(* Logix 5000 project; controller CLASE_1 Emulate 5570 rev 28.11; software revision 28.02; part 8 of 15 *)
(* tags used below, declared in another part *)
   Inp_PosFdbk : REAL;   // Position Feedback from Valve (in Raw Input units)
   Inp_OpenLS : BOOL;   // Valve Open Limit Switch 1=confirmed fully open
   Inp_ClosedLS : BOOL;   // Valve Closed Limit Switch 1=confirmed fully closed
   Inp_ActuatorFault : BOOL;   // Valve Actuator Fault (overload, etc.), 0=OK, 1=Fault)
   Inp_IntlkOK : BOOL;   // 1=Interlocks OK, Pulse Output Valve can be moved
   Inp_NBIntlkOK : BOOL;   // 1=Non-Bypassable Interlocks OK, Pulse Output Valve can be moved
   Inp_IOFault : BOOL;   // Input / Output Communication Status 0=OK, 1=fail
   Inp_Sim : BOOL;   // 1=I/O are being simulated, set output CV to 0.0, ignore I/O Fault
   Inp_OvrdCV : REAL;   // CV target in Override Mode (CV EU)
   Inp_Reset : BOOL;   // 1=Reset latched Alarms
   Cfg_ShedHold : BOOL;   // 1=Hold Output on Interlock or bad PV, 0=Go to Cfg_IntlkCV
   Cfg_ShedOnIOFault : BOOL;   // 1=Take shed action (hold or interlock CV) on I/O Fault
   Cfg_SkipRoCLim : BOOL;   // 1=Skip RoC Limiting in Intlk, Maint, Ovrd modes
   Cfg_SetTrack : BOOL;   // 1=PSets track OSets in Oper, OSets track PSets in Prog, 0=no tracking
   Cfg_SetTrackOvrdHand : BOOL;   // 1=Prog/Oper Settings track Override/Hand CV
   Cfg_HasOpenLS : BOOL;   // 1=Valve provides an Open Limit Switch signal
   Cfg_HasClosedLS : BOOL;   // 1=Valve provides a Closed Limit Switch signal
   Cfg_UseOpenLS : BOOL;   // 1=Valve Open LS should be used for open/closed status
   Cfg_UseClosedLS : BOOL;   // 1=Valve Closed LS should be used for open/closed status
   Cfg_LSFail : BOOL;   // 1=both switches ON=fail, 0=both switches OFF=fail
   Cfg_PCmdClear : ALIAS FOR Mode.Cfg_PCmdClear;
   Cfg_OvrdIntlk : BOOL;   // 1=Override ignores Bypassable Intlk; 0=always use Intlk
   Cfg_MinCV : REAL;   // Minimum CV (in CV EU, for limiting)
   Cfg_MaxCV : REAL;   // Maximum CV (in CV EU, for limiting)
   Cfg_MaxCVRoCInc : REAL;   // Maximum allowed CV Rate of Change (Increasing) Setting (EU/sec)
   Cfg_MaxCVRoCDec : REAL;   // Maximum allowed CV Rate of Change (Decreasing) Setting (EU/sec)
   Cfg_IntlkCV : REAL;   // CV (target in EU) when interlocked (if not Cfg_ShedHold)
   Cfg_CVEUMin : REAL;   // CV Minimum in Engineering Units (for scaling)
   Cfg_CVEUMax : REAL;   // CV Maximum in Engineering Units (for scaling)
   Cfg_CVRawMin : REAL;   // CV Minimum in I/O (raw) Units (for scaling)
   Cfg_CVRawMax : REAL;   // CV Maximum in I/O (raw) Units (for scaling)
   Cfg_FdbkRawMin : REAL;   // Position Feedback Minimum in raw input units (for scaling)
   Cfg_FdbkRawMax : REAL;   // Position Feedback Maximum in raw input units (for scaling)
   Cfg_CycleT : REAL;   // Open and Close Pulse Output overall period (s)
   Cfg_OpenRate : REAL;   // Rate at which valve moves when opening (CV EU/sec)
   Cfg_CloseRate : REAL;   // Rate at which valve moves when closing (CV EU/sec)
   Cfg_MaxOnT : REAL;   // Open and Close Pulse Output maximum ON time (s)
   Cfg_MinOnT : REAL;   // Open and Close Pulse Output minimum ON time (s)
   Cfg_BumpT : REAL;   // Time to bump valve open or closed (by Oper) when Fdbk Bad (sec)
   Cfg_Deadtime : REAL;   // Additional time on first pulse after stop or direction change
   Cfg_MaxClosedPos : REAL;   // Position above which valve is assumed open if limit switches not used
   PSet_CV : REAL;   // Program Setting of Controlled Variable (output) (CV EU)
   PSet_CVRoCLimInc : REAL;   // Program Setting of CV Rate of Change Limit, Increasing, (in EU/sec)
   PSet_CVRoCLimDec : REAL;   // Program Setting of CV Rate of Change Limit, Decreasing, (in EU/sec)
   PSet_Owner : DINT;   // Program Owner Request ID (non-zero) or Release (zero)
   OSet_CV : REAL;   // Operator Setting of Controlled Variable (output) (CV EU)
   OSet_CVRoCLimInc : REAL;   // Operator Setting of CV Rate of Change Limit, Increasing, (in EU/sec)
   OSet_CVRoCLimDec : REAL;   // Operator Setting of CV Rate of Change Limit, Decreasing, (in EU/sec)
   PCmd_Reset : BOOL;   // Program Command to Reset Alarms requiring Reset
   OCmd_BumpOpen : BOOL;   // Operator Command to bump valve open (avail. if Fdbk Bad)
   OCmd_BumpClose : BOOL;   // Operator Command to bump valve closed (avail. if Fdbk Bad)
   OCmd_Bypass : BOOL;   // Operator Command to Bypass all Bypassable Interlocks
   OCmd_Check : BOOL;   // Operator Command to Check (not bypass) all Interlocks
   MCmd_Disable : BOOL;   // Maintenance Command to Pulse Output Valve
   MCmd_Enable : BOOL;   // Maintenance Command to Enable Pulse Output Valve
   OCmd_Reset : BOOL;   // Operator Command to Reset all Alarms requiring Reset
   OCmd_ResetAckAll : BOOL;   // Operator Command to Reset all Alarms and latched Shed conditions
   Out_CV : REAL;   // CV Output in Raw (I/O Card) Units
   Val_Pos : REAL;   // Valve actual position from feedback (CV EU)
   Val_CVOut : REAL;   // Value of CV output (after clamping and ramping) (CV EU)
   Val_CVEUMin : REAL;   // Minimum of scaled range = MIN (Cfg_CVEUMin, Cfg_CVEUMax)
   Val_CVEUMax : REAL;   // Maximum of scaled range = MAX (Cfg_CVEUMin, Cfg_CVEUMax)
   SrcQ_IO : SINT;   // Source and Quality of primary I/O (enumeration)
   SrcQ : SINT;   // Source and Quality of primary Val/Sts (enumeration)
   Val_Fdbk : SINT;   // Device Feedback 0=Moving, 1=Closed, 2=Opened, 3=Limit Switch Failure
   Val_Sts : SINT;   // 0=AtTarget, 1=RampClose, 2=RampOpen, 3=Clamp@Min, 4=Clamp@Max, 5=BumpClose, 6=BumpOpen, 33=Disabled
   Val_Owner : DINT;   // Current Object Owner ID (0=not owned)
   Sts_CVInfNaN : BOOL;   // 1=Selected CV is Infinite or Not A Number (1.$, 1.#NaN)
   Sts_PosInfNaN : BOOL;   // 1=Inp_PosFdbk is Infinite or Not A Number (1.$, 1.#NaN)
   Sts_Ramping : BOOL;   // 1=CV is ramping to target
   Sts_Clamped : BOOL;   // 1=CV Set is clamped at CVMin or CVMax
   Sts_SkipRoCLim : BOOL;   // 1=Rate of Change Limiting was skipped this scan (Maint, Ovrd, Intlk, Hand)
   Sts_Active : BOOL;   // 1=CV is greater than Cfg_MaxClosedPos, show valve symbol as "opened"
   Sts_Available : BOOL;   // 1=Pulse Output Valve available for control by automation (Prog)
   Sts_Bypass : BOOL;   // 1=Bypassable Interlocks are Bypassed
   Sts_BypActive : BOOL;   // 1=Bypassing Active (Bypassed or Maintenance)
   Sts_Disabled : BOOL;   // 1=Output is Disabled
   Sts_LSFail : BOOL;   // 1=Limit Switch Overlap Failure
   Sts_NotRdy : BOOL;   // 1=Device Not Ready, see detail bits for reason
   Nrdy_Disabled : BOOL;   // 1=Device Not Ready: Device Disabled by Maintenance
   Nrdy_CfgErr : BOOL;   // 1=Device Not Ready: Configuration Error
   Nrdy_Intlk : BOOL;   // 1=Device Not Ready: Interlock Not OK
   Nrdy_IOFault : BOOL;   // 1=Device Not Ready: I/O Fault (Shed Requires Reset)
   Nrdy_NoMode : BOOL;   // 1=Device Not Ready: Device Logic Disabled / NO Mode
   Sts_MaintByp : BOOL;   // 1=Device has a Maintenance Bypass function active
   Sts_Err : BOOL;   // 1=Error in Config: see detail bits for reason
   Err_Limit : BOOL;   // 1=Error in Config: CV Limits swapped
   Err_EU : BOOL;   // 1=Error in Config: Scaled CV EU Min = Max
   Err_Raw : BOOL;   // 1=Error in Config: Raw Output Scaling Min = Max
   Err_Fdbk : BOOL;   // 1=Error in Config: Raw Feedback Scaling Min = Max
   Err_Timer : BOOL;   // 1=Error in Config: Invalid Timer Preset (use 0 to 2147483)
   Err_Alarm : BOOL;   // 1=Error in Config: Alarm Min On Time, Shelf Time, Severity
   Sts_Hand : ALIAS FOR Mode.Sts_Hand;
   Sts_Maint : ALIAS FOR Mode.Sts_Maint;
   Sts_Ovrd : ALIAS FOR Mode.Sts_Ovrd;
   Sts_Prog : ALIAS FOR Mode.Sts_Prog;
   Sts_Oper : ALIAS FOR Mode.Sts_Oper;
   Sts_IntlkTrip : ALIAS FOR IntlkTrip.Inp;   // 1=Status: CV held or forced by interlock NOT OK (1-shot)
   Sts_ActuatorFault : ALIAS FOR ActuatorFault.Inp;   // 1=Actuator Fault detected (input)
   Sts_IOFault : ALIAS FOR IOFault.Inp;   // 1=I/O Fault Status (0=OK, 1=Bad)
   Rdy_BumpOpen : BOOL;   // 1=Ready to receive OCmd_BumpOpen (enables HMI button)
   Rdy_BumpClose : BOOL;   // 1=Ready to receive OCmd_BumpClose (enables HMI button)
   Rdy_Bypass : BOOL;   // 1=Ready to receive OCmd_Bypass (enables HMI button)
   Rdy_Check : BOOL;   // 1=Ready to receive OCmd_Check (enables HMI button)
   Rdy_Disable : BOOL;   // 1=Ready to receive MCmd_Disable (enables HMI button)
   Rdy_Enable : BOOL;   // 1=Ready to receive MCmd_Enable (enables HMI button)
   Rdy_CV : BOOL;   // 1=Ready to receive OSet_CV (enables data entry field)
   Rdy_CVRoCLimInc : BOOL;   // 1=Ready to receive OSet_CVRoCLimInc (enables data entry field)
   Rdy_CVRoCLimDec : BOOL;   // 1=Ready to receive OSet_CVRoCLimDec (enables data entry field)
   P_ValveC : BOOL;   // Unique Parameter Name for auto - discovery
   Mode : P_Mode;   // Pulse Output Valve Mode Selection
   IOFault : P_Alarm;   // I/O Fault Alarm
   IntlkTrip : P_Alarm;   // Interlock Trip Alarm
   Cfg_Tag : STRING_20;   // Tagname for display on HMI
   Cfg_Label : STRING_20;   // Label for graphic symbol displayed on HMI
   Cfg_Desc : STRING_40;   // Description for display on HMI
   Wrk_Bypass : BOOL;   // Internal Bypassable Interlocks are Bypassed flag
   Wrk_Disabled : BOOL;   // Internal Pulse Output Valve Disabled status
   Cfg_EU : STRING_8;   // Engineering Units for display on HMI
   Wrk_CV : REAL;   // Working copy of Speed Reference (for limiting)
   Wrk_CVRoCLimInc : REAL;   // Selected CV Rate of Change Limit Increasing
   Wrk_CVSet : REAL;   // Final selected CV to feed to RoC Limiter
   Wrk_CVOut : REAL;   // Working value of CV after Rate Limiting
   Wrk_IntlkTripONS : BOOL;   // Interlock Tripped This Scan
   Wrk_ScanTime : REAL;   // Seconds since previous scan
   Wrk_StepInc : REAL;   // Amount to increase CV (to valve pulse logic) this scan for rate limiting
   Wrk_ScanT : TIMER;   // Scan Timer (milliseconds, always runs)
   ActuatorFault : P_Alarm;   // Actuator Fault Alarm (based on Actuator Fault Input)
   Wrk_RealChkDINT : DINT;   // REAL tag bit pattern as a DINT to check for Inf / NaN
   Wrk_Close : BOOL;   // Internal Close output -- before Sim
   Wrk_Open : BOOL;   // Internal Open output -- before Sim
   Wrk_CycleT : TIMER;   // Overall Cycle Timer for pulsed outputs
   Wrk_OKtoOpen : BOOL;   // OK to pulse Out_Open
   Wrk_OKtoClose : BOOL;   // OK to pulse Out_Close
   Wrk_OpenTime : REAL;   // Time to pulse Out_Open
   Wrk_CycleT_ms : DINT;   // Cycle Time in milliseconds (preset)
   Wrk_CloseTime : REAL;   // Time to pulse Out_Close
   Inf_Type : STRING_16;   // Must contain AOI name, used for HMI and Information S/W
   Wrk_OpenFdbk : BOOL;   // 1=LS Feedback shows valve confirmed open
   Wrk_ClosedFdbk : BOOL;   // 1=LS Feedback shows valve confirmed closed
   Wrk_StepDec : REAL;   // Amount to decrease CV (to valve pulse logic) this scan for rate limiting
   Wrk_CVRoCLimDec : REAL;   // Selected CV Rate of Change Limit Decreasing
   Wrk_BumpClose : BOOL;   // Operator Bump Close requested
   Wrk_BumpOpen : BOOL;   // Operator Bump Open requested
   Wrk_BumpingOpen : BOOL;   // Operator Bump Open actively pulsing Out_Open
   Wrk_BumpingClose : BOOL;   // Operator Bump Close actively pulsing Out_Close
   Inf_Lib : STRING_12;   // Display Library for Faceplate call-up
   Cfg_CVNavTag : STRING_NavTag;   // Tagname for destination of CV Navigation button
   Wrk_ShedIntlkCV : BOOL;   // Output CV being held at Interlock value
   Wrk_ShedHold : BOOL;   // Output CV being held at last good value
(* P_ValveC, continued *)

ROUTINE Logic   (* ladder *)
// Normal Scan: control Analog Output
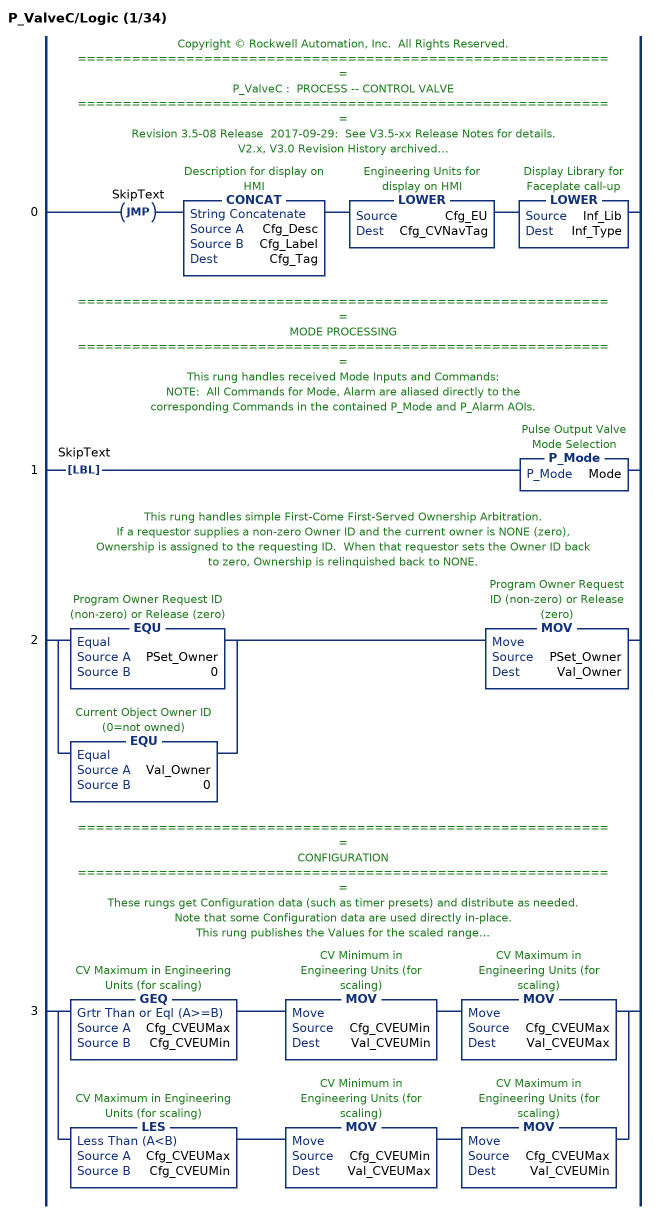
   // Copyright © Rockwell Automation, Inc.  All Rights Reserved.
   // ============================================================
   // P_ValveC :  PROCESS -- CONTROL VALVE
   // ============================================================
   // Revision 3.5-08 Release  2017-09-29:  See V3.5-xx Release Notes for details.
   // V2.x, V3.0 Revision History archived.
   // V3.1-00  2014-07-22:  Modified to use P_Alarm, P_Mode V3.1; added
   // Not Ready reason bits (Nrdy_Xxxxx), source/quality values (SrcQ).
   // Modified to consistently use alias tag names.  Added check for
   // Err_Fdbk on scaling of position feedback.
   // V3.1-01  2014-09-03:  Corrections to Nrdy_ resets. Modified logic for
   // Err_Fdbk. Using P_Alarm, P_Mode V3.1-01.
   // V3.1-02  2014-09-30:  Unchanged, but using P_Alarm V3.1-02.
   // V3.1-03  2015-01-21:  Corrected Maintenance Bypass indication for limit switches.
   // Modified to prevent output pulsing on additional fault conditions.
   //  Modified to show Val_Sts = 1 or 2 when moving via pulsing.
   // V3.1-04 Patch01  2015-09-25: Modified Err_Fdbk, Err_Raw, handling of Cfg_CycleT.
   // V3.5-01  2016-01-29:  Unchanged, but using P_Alarm V3.5-01.
   // V3.5-03 Patch01  2016-07-06:  Modified logic which triggers IntlkTrip status/alarm.
   // V3.5-05  2016-12-16:   Changed Nav Tags to user-defined STRING_NavTag type.
   // V3.5-08  2017-09-29:  Modified CV Rate of Change handling for limits = 0.0 (unlimited).
   // ============================================================
   // This Instruction controls a Pulse Output Valve with
   // analog position feedback and provides:
   // *  Program and Operator entry of target position in Percent Open
   // *  Ramping of position to target at specified Rate of Change (%/sec)
   // *  Scaling of Position Feedback input from Raw (I/O card) Units to percent
   // *  Monitoring of Interlock conditions which cause output to shed
   // *  Configurable shed to HOLD or to configured position
   // *  Monitoring of I/O communication faults
   // *  Alarms for Interlock Trip, Actuator Fault, I/O Fault
   // *  Opened, Closed status based on limit switches (if provided),
   // or based on Position Feedback and a configured threshold.
   // *  "Available" status for use by automation logic to know whether valve
   //       can be controlled by other objects.
   // Modes are provided by a P_Mode AOI instance.
   // Alarms are provided by P_Alarm AOI instances.
   // Modes of operation: Operator, Program, Override, Maintenance, Hand
   // ============================================================
   // SHOW LOCAL STRINGS
   // ============================================================
   // The STRINGs containing the text associated with each instance of this
   // instruction cannot be Input or Output Parameters, because STRINGs are not
   //  'atomic' types. (Inputs and Outputs must be SINT, INT, DINT, REAL, or BOOL.)
   // In order to make it easier to find and configure these STRINGs, this rung
   // was added.  THE JMP (and the LBL on the following rung)
   // MUST NOT BE REMOVED!!!
   // To view the STRINGs, go to the instruction instance (in LD or FBD), RIGHT-click
   // to bring up the context menu and select "Open Instruction Logic".
   // This rung will appear with the STRING values for the selected instance.
   // You may double-click the STRING values here to modify them as well.
   // #####  V3.1-00  2014-07-15: Added Cfg_CVNavTag to displayed strings  #####
   0: JMP(SkipText)CONCAT(Cfg_Desc,Cfg_Label,Cfg_Tag)LOWER(Cfg_EU,Cfg_CVNavTag)LOWER(Inf_Lib,Inf_Type);
   // ============================================================
   // MODE PROCESSING
   // ============================================================
   // This rung handles received Mode Inputs and Commands:
   // NOTE:  All Commands for Mode, Alarm are aliased directly to the
   // corresponding Commands in the contained P_Mode and P_Alarm AOIs.
   1: LBL(SkipText)P_Mode(Mode);
   // This rung handles simple First-Come First-Served Ownership Arbitration.
   // If a requestor supplies a non-zero Owner ID and the current owner is NONE (zero),
   // Ownership is assigned to the requesting ID.  When that requestor sets the Owner ID back
   // to zero, Ownership is relinquished back to NONE.
   2: [EQU(PSet_Owner,0) ,EQU(Val_Owner,0) ]MOV(PSet_Owner,Val_Owner);
   // ============================================================
   // CONFIGURATION
   // ============================================================
   // These rungs get Configuration data (such as timer presets) and distribute as needed.
   // Note that some Configuration data are used directly in-place.
   // This rung publishes the Values for the scaled range.
   // If this instruction is reverse scaled by reversing the scaled (EU) min and max configurations,
   // the values are swapped so the the EUMax Value is always greater than the EUMin Value.
   // This makes the HMI bargraph and trend coding easier, and provides values
   // that can be pinned to the CV EU configuration of a PID, so the AOut and PID ranges are in lockstep.
   3: [GEQ(Cfg_CVEUMax,Cfg_CVEUMin) MOV(Cfg_CVEUMin,Val_CVEUMin) MOV(Cfg_CVEUMax,Val_CVEUMax) ,LES(Cfg_CVEUMax,Cfg_CVEUMin) MOV(Cfg_CVEUMin,Val_CVEUMax) MOV(Cfg_CVEUMax,Val_CVEUMin) ];
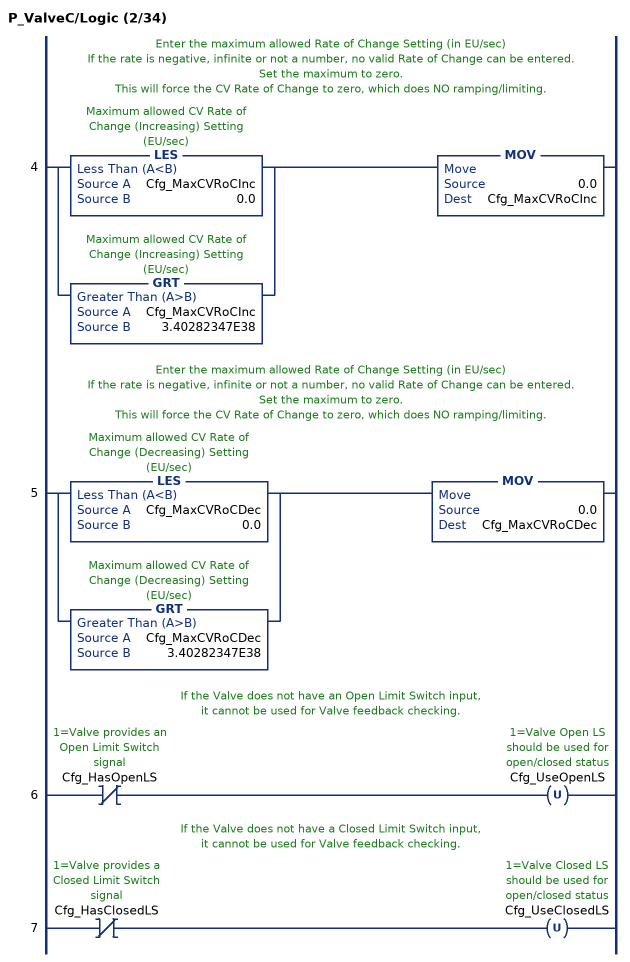
   // Enter the maximum allowed Rate of Change Setting (in EU/sec)
   // If the rate is negative, infinite or not a number, no valid Rate of Change can be entered.  Set the maximum to zero.
   // This will force the CV Rate of Change to zero, which does NO ramping/limiting.
   4: [LES(Cfg_MaxCVRoCInc,0.0) ,GRT(Cfg_MaxCVRoCInc,3.40282347E38) ]MOV(0.0,Cfg_MaxCVRoCInc);
   // Enter the maximum allowed Rate of Change Setting (in EU/sec)
   // If the rate is negative, infinite or not a number, no valid Rate of Change can be entered.  Set the maximum to zero.
   // This will force the CV Rate of Change to zero, which does NO ramping/limiting.
   5: [LES(Cfg_MaxCVRoCDec,0.0) ,GRT(Cfg_MaxCVRoCDec,3.40282347E38) ]MOV(0.0,Cfg_MaxCVRoCDec);
   // If the Valve does not have an Open Limit Switch input,
   // it cannot be used for Valve feedback checking.
   6: XIO(Cfg_HasOpenLS)OTU(Cfg_UseOpenLS);
   // If the Valve does not have a Closed Limit Switch input,
   // it cannot be used for Valve feedback checking.
   7: XIO(Cfg_HasClosedLS)OTU(Cfg_UseClosedLS);
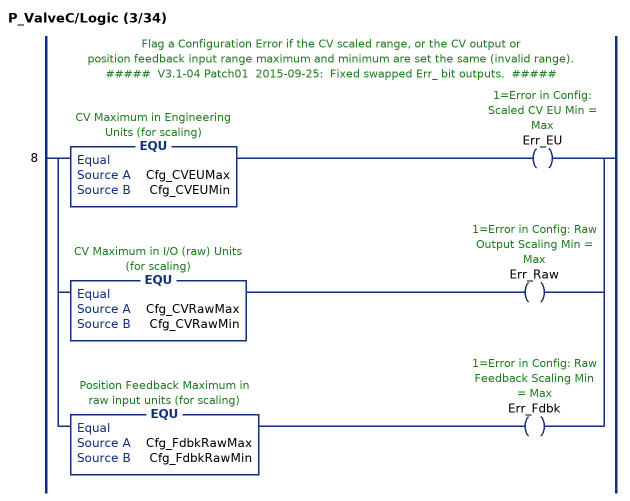
   // Flag a Configuration Error if the CV scaled range, or the CV output or
   // position feedback input range maximum and minimum are set the same (invalid range).
   // #####  V3.1-04 Patch01  2015-09-25:  Fixed swapped Err_ bit outputs.  #####
   8: [EQU(Cfg_CVEUMax,Cfg_CVEUMin) OTE(Err_EU) ,EQU(Cfg_CVRawMax,Cfg_CVRawMin) OTE(Err_Raw) ,EQU(Cfg_FdbkRawMax,Cfg_FdbkRawMin) OTE(Err_Fdbk) ];
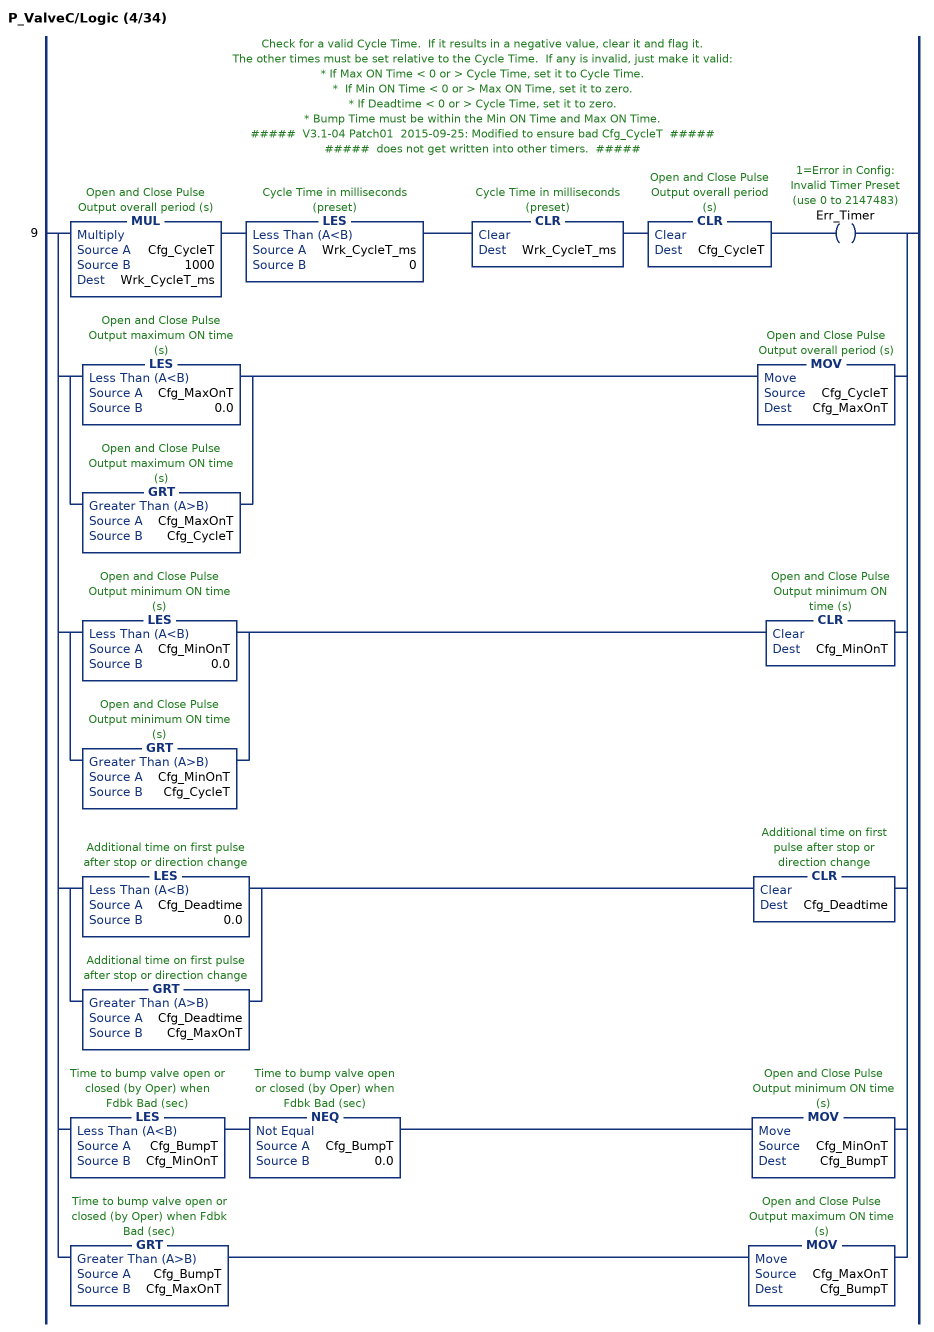
   // Check for a valid Cycle Time.  If it results in a negative value, clear it and flag it.
   // The other times must be set relative to the Cycle Time.  If any is invalid, just make it valid:
   // * If Max ON Time < 0 or > Cycle Time, set it to Cycle Time.
   // *  If Min ON Time < 0 or > Max ON Time, set it to zero.
   // * If Deadtime < 0 or > Cycle Time, set it to zero.
   // * Bump Time must be within the Min ON Time and Max ON Time.
   // #####  V3.1-04 Patch01  2015-09-25: Modified to ensure bad Cfg_CycleT  #####
   // #####  does not get written into other timers.  #####
   9: [MUL(Cfg_CycleT,1000,Wrk_CycleT_ms) LES(Wrk_CycleT_ms,0) CLR(Wrk_CycleT_ms) CLR(Cfg_CycleT) OTE(Err_Timer) ,[LES(Cfg_MaxOnT,0.0) ,GRT(Cfg_MaxOnT,Cfg_CycleT) ] MOV(Cfg_CycleT,Cfg_MaxOnT) ,[LES(Cfg_MinOnT,0.0) ,GRT(Cfg_MinOnT,Cfg_CycleT) ] CLR(Cfg_MinOnT) ,[LES(Cfg_Deadtime,0.0) ,GRT(Cfg_Deadtime,Cfg_MaxOnT) ] CLR(Cfg_Deadtime) ,LES(Cfg_BumpT,Cfg_MinOnT) NEQ(Cfg_BumpT,0.0) MOV(Cfg_MinOnT,Cfg_BumpT) ,GRT(Cfg_BumpT,Cfg_MaxOnT) MOV(Cfg_MaxOnT,Cfg_BumpT) ];
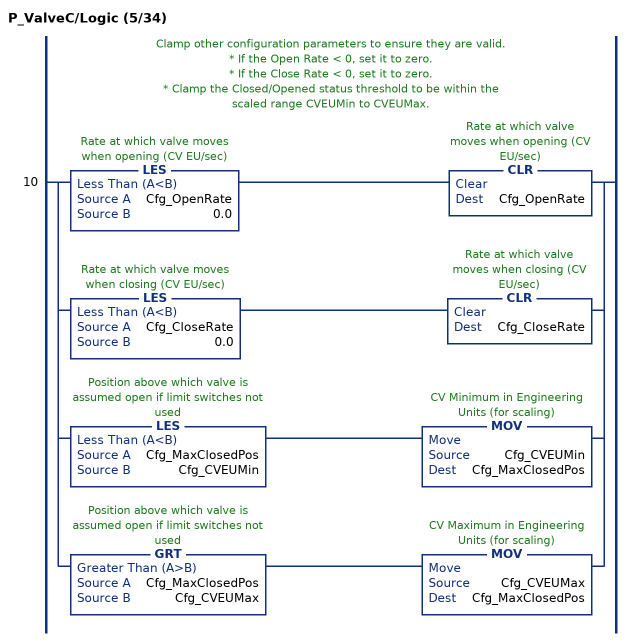
   // Clamp other configuration parameters to ensure they are valid.
   // * If the Open Rate < 0, set it to zero.
   // * If the Close Rate < 0, set it to zero.
   // * Clamp the Closed/Opened status threshold to be within the
   // scaled range CVEUMin to CVEUMax.
   10: [LES(Cfg_OpenRate,0.0) CLR(Cfg_OpenRate) ,LES(Cfg_CloseRate,0.0) CLR(Cfg_CloseRate) ,LES(Cfg_MaxClosedPos,Cfg_CVEUMin) MOV(Cfg_CVEUMin,Cfg_MaxClosedPos) ,GRT(Cfg_MaxClosedPos,Cfg_CVEUMax) MOV(Cfg_CVEUMax,Cfg_MaxClosedPos) ];
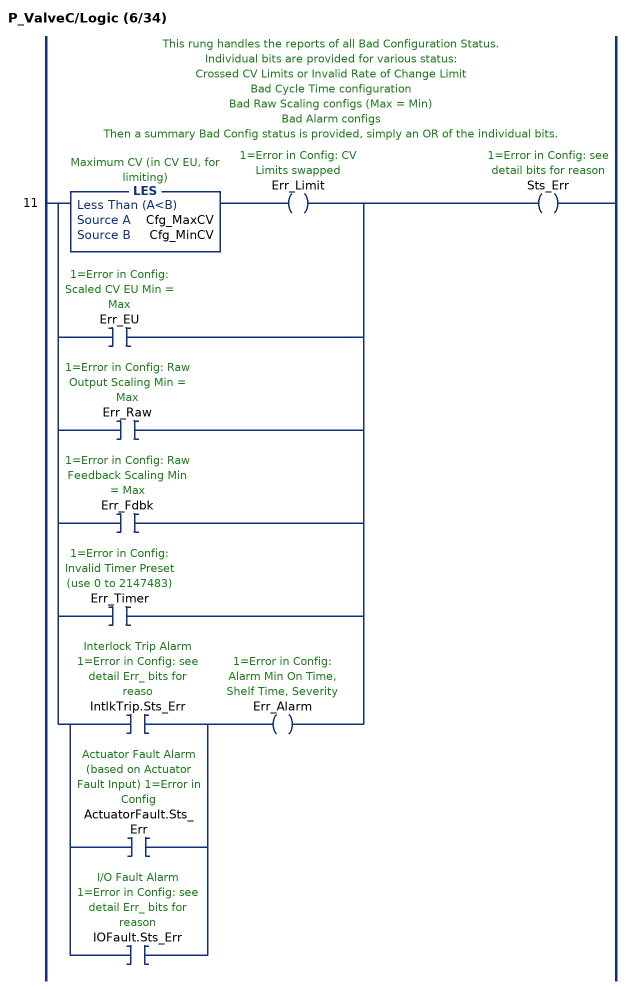
   // This rung handles the reports of all Bad Configuration Status.
   // Individual bits are provided for various status:
   // Crossed CV Limits or Invalid Rate of Change Limit
   // Bad Cycle Time configuration
   // Bad Raw Scaling configs (Max = Min)
   // Bad Alarm configs
   // Then a summary Bad Config status is provided, simply an OR of the individual bits.
   11: [LES(Cfg_MaxCV,Cfg_MinCV) OTE(Err_Limit) ,XIC(Err_EU) ,XIC(Err_Raw) ,XIC(Err_Fdbk) ,XIC(Err_Timer) ,[XIC(IntlkTrip.Sts_Err) ,XIC(ActuatorFault.Sts_Err) ,XIC(IOFault.Sts_Err) ] OTE(Err_Alarm) ]OTE(Sts_Err);
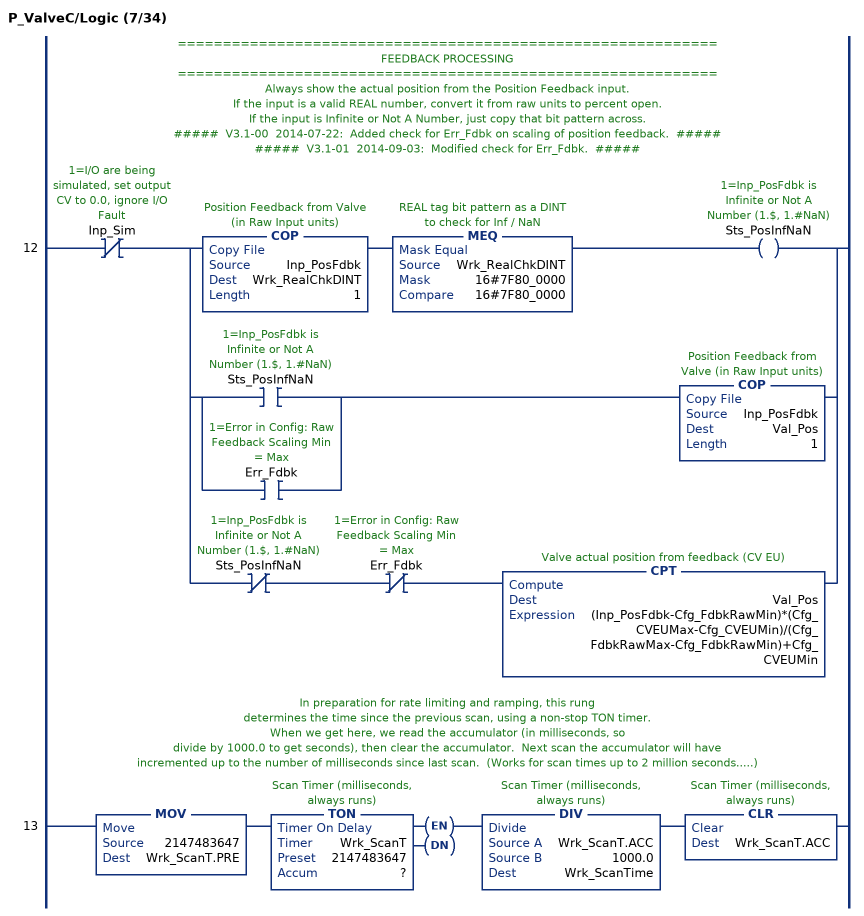
   // ============================================================
   // FEEDBACK PROCESSING
   // ============================================================
   // Always show the actual position from the Position Feedback input.
   // If the input is a valid REAL number, convert it from raw units to percent open.
   // If the input is Infinite or Not A Number, just copy that bit pattern across.
   // #####  V3.1-00  2014-07-22:  Added check for Err_Fdbk on scaling of position feedback.  #####
   // #####  V3.1-01  2014-09-03:  Modified check for Err_Fdbk.  #####
   12: XIO(Inp_Sim)[COP(Inp_PosFdbk,Wrk_RealChkDINT,1) MEQ(Wrk_RealChkDINT,16#7F80_0000,16#7F80_0000) OTE(Sts_PosInfNaN) ,[XIC(Sts_PosInfNaN) ,XIC(Err_Fdbk) ] COP(Inp_PosFdbk,Val_Pos,1) ,XIO(Sts_PosInfNaN) XIO(Err_Fdbk) CPT(Val_Pos,(Inp_PosFdbk-Cfg_FdbkRawMin)*(Cfg_CVEUMax-Cfg_CVEUMin)/(Cfg_FdbkRawMax-Cfg_FdbkRawMin)+Cfg_CVEUMin) ];
   // In preparation for rate limiting and ramping, this rung
   // determines the time since the previous scan, using a non-stop TON timer.
   // When we get here, we read the accumulator (in milliseconds, so
   // divide by 1000.0 to get seconds), then clear the accumulator.  Next scan the accumulator will have
   // incremented up to the number of milliseconds since last scan.  (Works for scan times up to 2 million seconds.....)
   13: MOV(2147483647,Wrk_ScanT.PRE)TON(Wrk_ScanT,?,?)DIV(Wrk_ScanT.ACC,1000.0,Wrk_ScanTime)CLR(Wrk_ScanT.ACC);
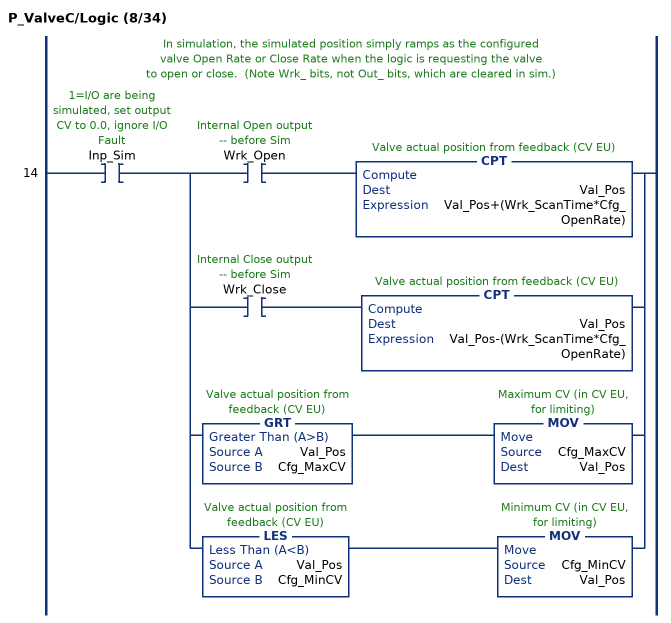
   // In simulation, the simulated position simply ramps as the configured
   // valve Open Rate or Close Rate when the logic is requesting the valve
   // to open or close.  (Note Wrk_ bits, not Out_ bits, which are cleared in sim.)
   14: XIC(Inp_Sim)[XIC(Wrk_Open) CPT(Val_Pos,Val_Pos+(Wrk_ScanTime*Cfg_OpenRate)) ,XIC(Wrk_Close) CPT(Val_Pos,Val_Pos-(Wrk_ScanTime*Cfg_OpenRate)) ,GRT(Val_Pos,Cfg_MaxCV) MOV(Cfg_MaxCV,Val_Pos) ,LES(Val_Pos,Cfg_MinCV) MOV(Cfg_MinCV,Val_Pos) ];
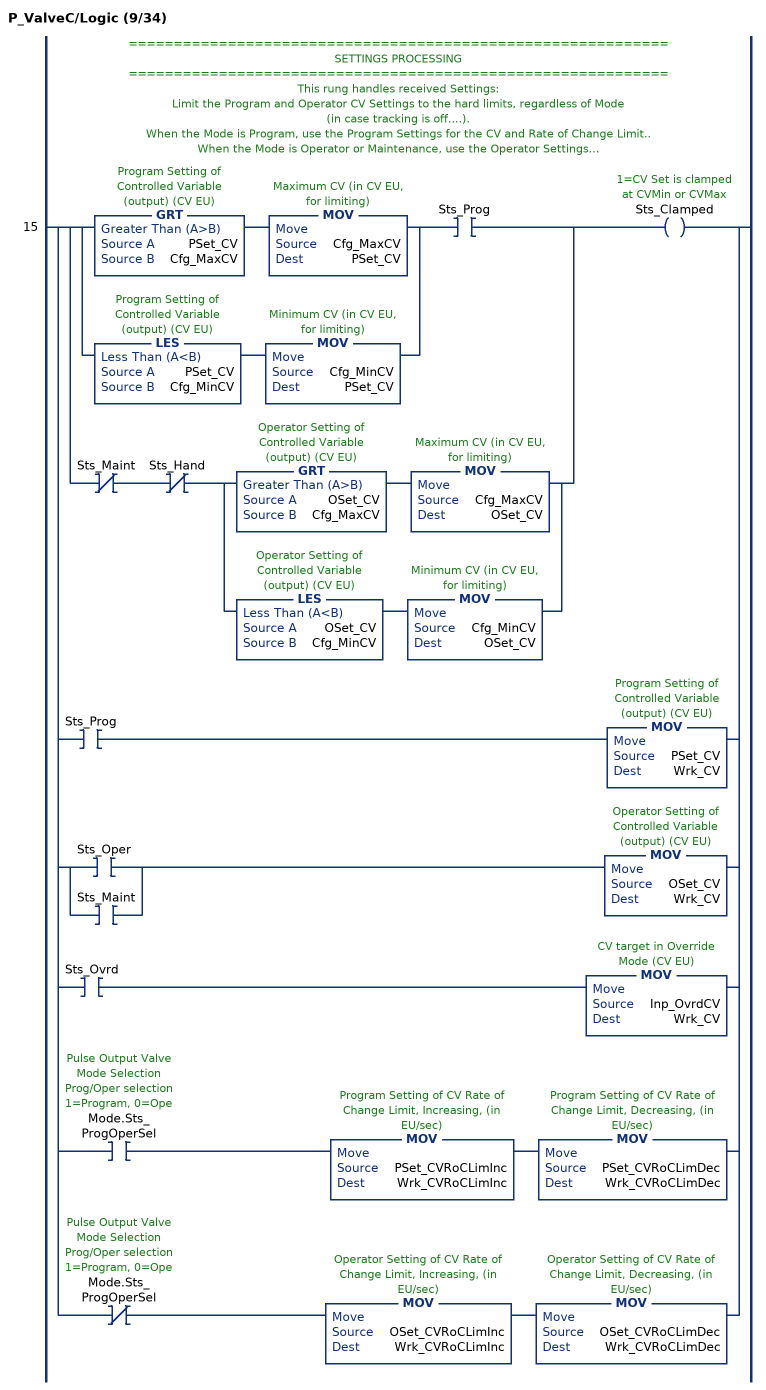
   // ============================================================
   // SETTINGS PROCESSING
   // ============================================================
   // This rung handles received Settings:
   // Limit the Program and Operator CV Settings to the hard limits, regardless of Mode
   // (in case tracking is off....).
   // When the Mode is Program, use the Program Settings for the CV and Rate of Change Limit..
   // When the Mode is Operator or Maintenance, use the Operator Settings.
   // When the Mode is Override, use the Override CV input for the CV.
   15: [[[GRT(PSet_CV,Cfg_MaxCV) MOV(Cfg_MaxCV,PSet_CV) ,LES(PSet_CV,Cfg_MinCV) MOV(Cfg_MinCV,PSet_CV) ] XIC(Sts_Prog) ,XIO(Sts_Maint) XIO(Sts_Hand) [GRT(OSet_CV,Cfg_MaxCV) MOV(Cfg_MaxCV,OSet_CV) ,LES(OSet_CV,Cfg_MinCV) MOV(Cfg_MinCV,OSet_CV) ] ] OTE(Sts_Clamped) ,XIC(Sts_Prog) MOV(PSet_CV,Wrk_CV) ,[XIC(Sts_Oper) ,XIC(Sts_Maint) ] MOV(OSet_CV,Wrk_CV) ,XIC(Sts_Ovrd) MOV(Inp_OvrdCV,Wrk_CV) ,XIC(Mode.Sts_ProgOperSel) MOV(PSet_CVRoCLimInc,Wrk_CVRoCLimInc) MOV(PSet_CVRoCLimDec,Wrk_CVRoCLimDec) ,XIO(Mode.Sts_ProgOperSel) MOV(OSet_CVRoCLimInc,Wrk_CVRoCLimInc) MOV(OSet_CVRoCLimDec,Wrk_CVRoCLimDec) ];
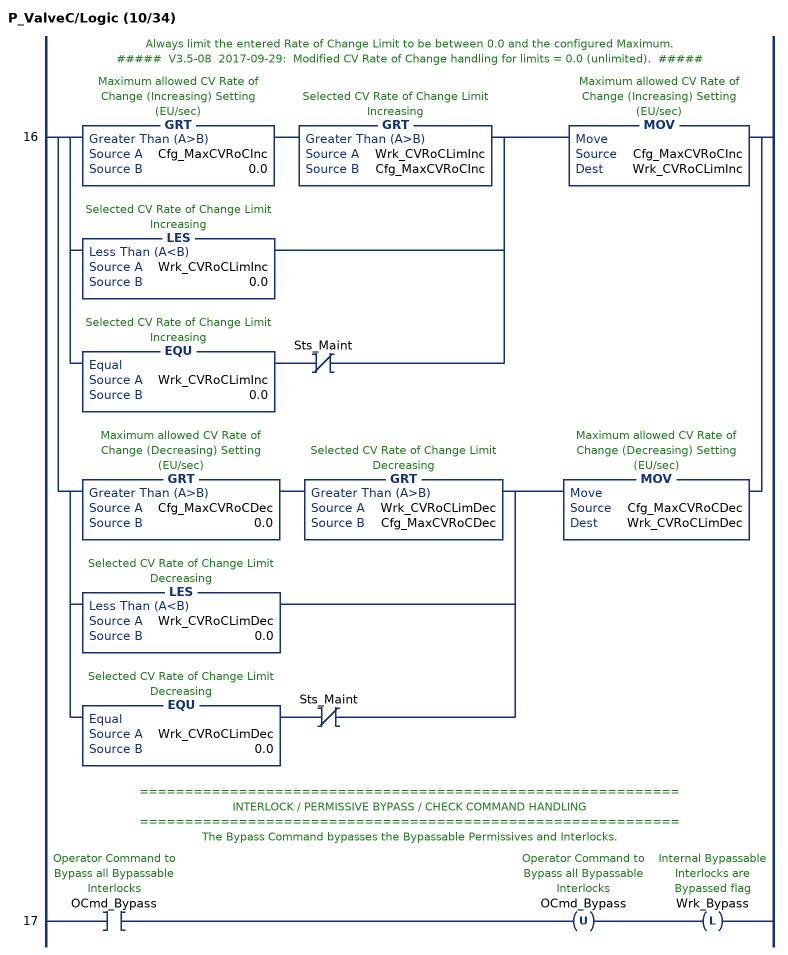
   // Always limit the entered Rate of Change Limit to be between 0.0 and the configured Maximum.
   // #####  V3.5-08  2017-09-29:  Modified CV Rate of Change handling for limits = 0.0 (unlimited).  #####
   16: [[GRT(Cfg_MaxCVRoCInc,0.0) GRT(Wrk_CVRoCLimInc,Cfg_MaxCVRoCInc) ,LES(Wrk_CVRoCLimInc,0.0) ,EQU(Wrk_CVRoCLimInc,0.0) XIO(Sts_Maint) ] MOV(Cfg_MaxCVRoCInc,Wrk_CVRoCLimInc) ,[GRT(Cfg_MaxCVRoCDec,0.0) GRT(Wrk_CVRoCLimDec,Cfg_MaxCVRoCDec) ,LES(Wrk_CVRoCLimDec,0.0) ,EQU(Wrk_CVRoCLimDec,0.0) XIO(Sts_Maint) ] MOV(Cfg_MaxCVRoCDec,Wrk_CVRoCLimDec) ];
   // ============================================================
   // INTERLOCK / PERMISSIVE BYPASS / CHECK COMMAND HANDLING
   // ============================================================
   // The Bypass Command bypasses the Bypassable Permissives and Interlocks.
   17: XIC(OCmd_Bypass)OTU(OCmd_Bypass)OTL(Wrk_Bypass);
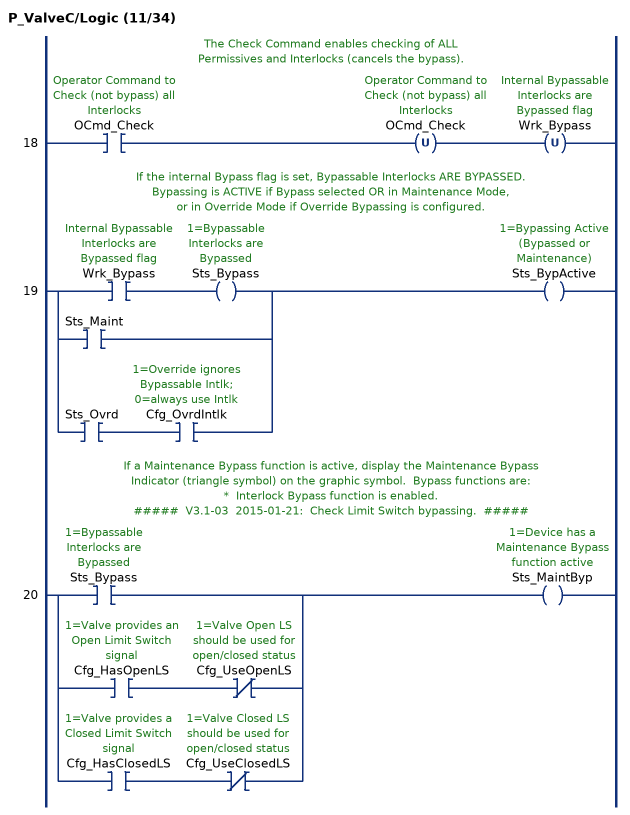
   // The Check Command enables checking of ALL
   // Permissives and Interlocks (cancels the bypass).
   18: XIC(OCmd_Check)OTU(OCmd_Check)OTU(Wrk_Bypass);
   // If the internal Bypass flag is set, Bypassable Interlocks ARE BYPASSED.
   // Bypassing is ACTIVE if Bypass selected OR in Maintenance Mode,
   // or in Override Mode if Override Bypassing is configured.
   19: [XIC(Wrk_Bypass) OTE(Sts_Bypass) ,XIC(Sts_Maint) ,XIC(Sts_Ovrd) XIC(Cfg_OvrdIntlk) ]OTE(Sts_BypActive);
   // If a Maintenance Bypass function is active, display the Maintenance Bypass
   // Indicator (triangle symbol) on the graphic symbol.  Bypass functions are:
   // *  Interlock Bypass function is enabled.
   // #####  V3.1-03  2015-01-21:  Check Limit Switch bypassing.  #####
   20: [XIC(Sts_Bypass) ,XIC(Cfg_HasOpenLS) XIO(Cfg_UseOpenLS) ,XIC(Cfg_HasClosedLS) XIO(Cfg_UseClosedLS) ]OTE(Sts_MaintByp);
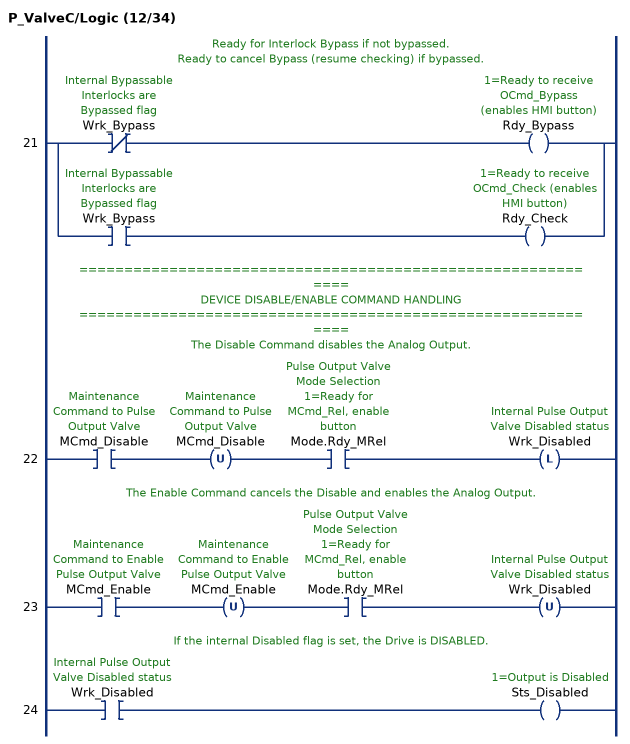
   // Ready for Interlock Bypass if not bypassed.
   // Ready to cancel Bypass (resume checking) if bypassed.
   21: [XIO(Wrk_Bypass) OTE(Rdy_Bypass) ,XIC(Wrk_Bypass) OTE(Rdy_Check) ];
   // ============================================================
   // DEVICE DISABLE/ENABLE COMMAND HANDLING
   // ============================================================
   // The Disable Command disables the Analog Output.
   22: XIC(MCmd_Disable)OTU(MCmd_Disable)XIC(Mode.Rdy_MRel)OTL(Wrk_Disabled);
   // The Enable Command cancels the Disable and enables the Analog Output.
   23: XIC(MCmd_Enable)OTU(MCmd_Enable)XIC(Mode.Rdy_MRel)OTU(Wrk_Disabled);
   // If the internal Disabled flag is set, the Drive is DISABLED.
   24: XIC(Wrk_Disabled)OTE(Sts_Disabled);
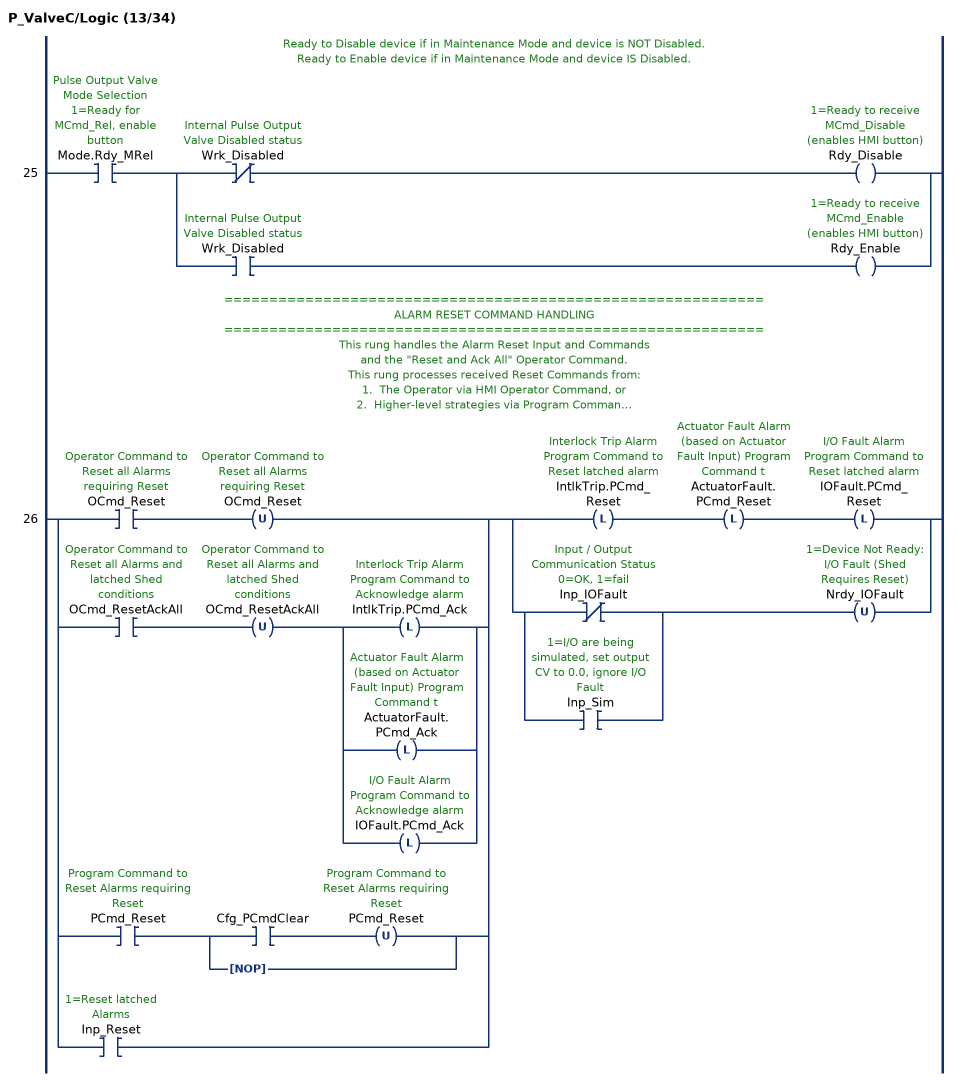
   // Ready to Disable device if in Maintenance Mode and device is NOT Disabled.
   // Ready to Enable device if in Maintenance Mode and device IS Disabled.
   25: XIC(Mode.Rdy_MRel)[XIO(Wrk_Disabled) OTE(Rdy_Disable) ,XIC(Wrk_Disabled) OTE(Rdy_Enable) ];
   // ============================================================
   // ALARM RESET COMMAND HANDLING
   // ============================================================
   // This rung handles the Alarm Reset Input and Commands
   // and the "Reset and Ack All" Operator Command.
   // This rung processes received Reset Commands from:
   // 1.  The Operator via HMI Operator Command, or
   // 2.  Higher-level strategies via Program Command
   // 3.  Pushbuttons or other block via Input
   // and forwards the Reset to ALL Alarms and latched Shed conditions.
   // #####  V3.1-00  2014-07-22: Added Not Ready reason bits (Nrdy_xxx)  #####
   // #####  V3.1-01  2014-09-03:  Corrections to Nrdy_ trip and reset logic.  #####
   26: [XIC(OCmd_Reset) OTU(OCmd_Reset) ,XIC(OCmd_ResetAckAll) OTU(OCmd_ResetAckAll) [OTL(IntlkTrip.PCmd_Ack) ,OTL(ActuatorFault.PCmd_Ack) ,OTL(IOFault.PCmd_Ack) ] ,XIC(PCmd_Reset) [XIC(Cfg_PCmdClear) OTU(PCmd_Reset) ,NOP() ] ,XIC(Inp_Reset) ][OTL(IntlkTrip.PCmd_Reset) OTL(ActuatorFault.PCmd_Reset) OTL(IOFault.PCmd_Reset) ,[XIO(Inp_IOFault) ,XIC(Inp_Sim) ] OTU(Nrdy_IOFault) ];
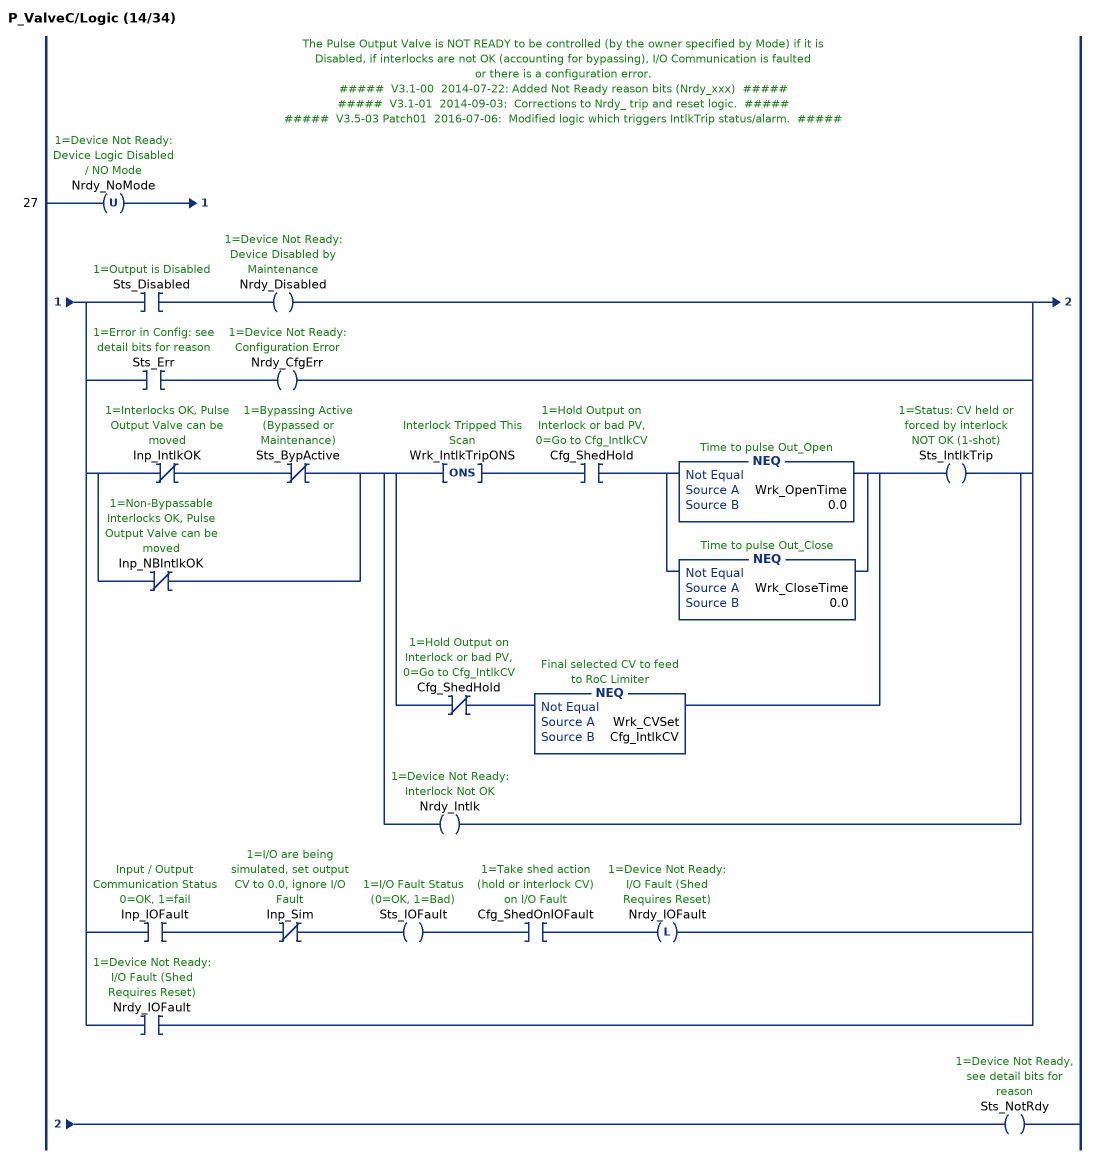
   // The Pulse Output Valve is NOT READY to be controlled (by the owner specified by Mode) if it is
   // Disabled, if interlocks are not OK (accounting for bypassing), I/O Communication is faulted
   // or there is a configuration error.
   // #####  V3.1-00  2014-07-22: Added Not Ready reason bits (Nrdy_xxx)  #####
   // #####  V3.1-01  2014-09-03:  Corrections to Nrdy_ trip and reset logic.  #####
   // #####  V3.5-03 Patch01  2016-07-06:  Modified logic which triggers IntlkTrip status/alarm.  #####
   27: OTU(Nrdy_NoMode)[XIC(Sts_Disabled) OTE(Nrdy_Disabled) ,XIC(Sts_Err) OTE(Nrdy_CfgErr) ,[XIO(Inp_IntlkOK) XIO(Sts_BypActive) ,XIO(Inp_NBIntlkOK) ] [[ONS(Wrk_IntlkTripONS) XIC(Cfg_ShedHold) [NEQ(Wrk_OpenTime,0.0) ,NEQ(Wrk_CloseTime,0.0) ] ,XIO(Cfg_ShedHold) NEQ(Wrk_CVSet,Cfg_IntlkCV) ] OTE(Sts_IntlkTrip) ,OTE(Nrdy_Intlk) ] ,XIC(Inp_IOFault) XIO(Inp_Sim) OTE(Sts_IOFault) XIC(Cfg_ShedOnIOFault) OTL(Nrdy_IOFault) ,XIC(Nrdy_IOFault) ]OTE(Sts_NotRdy);
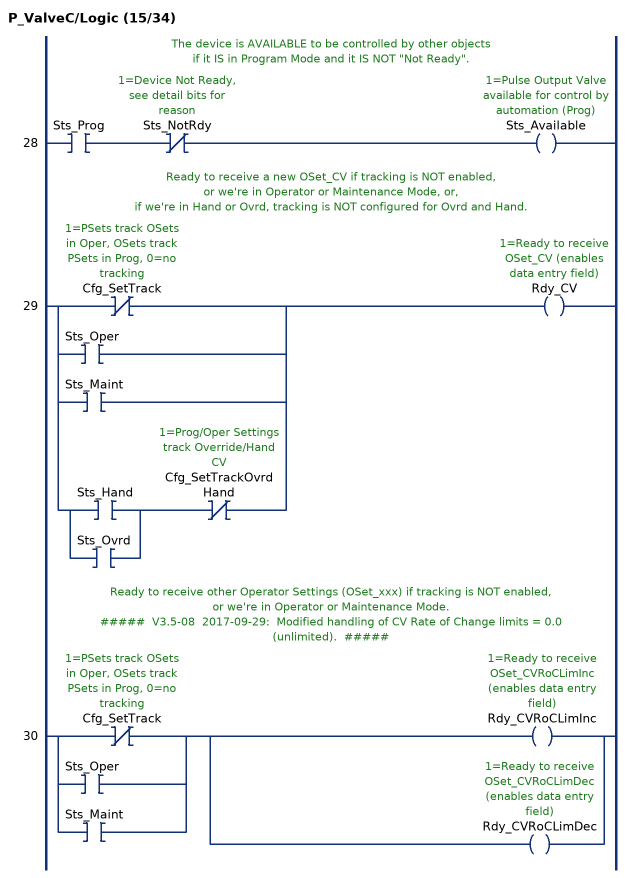
   // The device is AVAILABLE to be controlled by other objects
   // if it IS in Program Mode and it IS NOT "Not Ready".
   28: XIC(Sts_Prog)XIO(Sts_NotRdy)OTE(Sts_Available);
   // Ready to receive a new OSet_CV if tracking is NOT enabled,
   // or we're in Operator or Maintenance Mode, or,
   // if we're in Hand or Ovrd, tracking is NOT configured for Ovrd and Hand.
   29: [XIO(Cfg_SetTrack) ,XIC(Sts_Oper) ,XIC(Sts_Maint) ,[XIC(Sts_Hand) ,XIC(Sts_Ovrd) ] XIO(Cfg_SetTrackOvrdHand) ]OTE(Rdy_CV);
   // Ready to receive other Operator Settings (OSet_xxx) if tracking is NOT enabled,
   // or we're in Operator or Maintenance Mode.
   // #####  V3.5-08  2017-09-29:  Modified handling of CV Rate of Change limits = 0.0 (unlimited).  #####
   30: [XIO(Cfg_SetTrack) ,XIC(Sts_Oper) ,XIC(Sts_Maint) ][OTE(Rdy_CVRoCLimInc) ,OTE(Rdy_CVRoCLimDec) ];
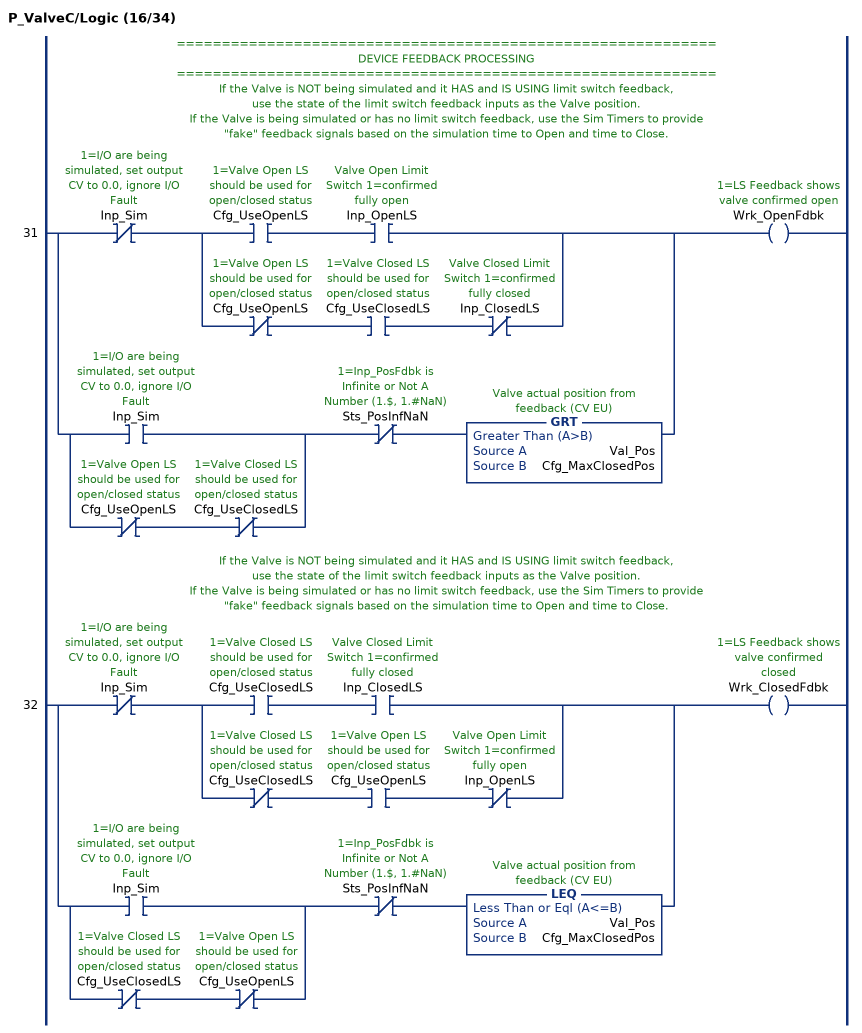
   // ============================================================
   // DEVICE FEEDBACK PROCESSING
   // ============================================================
   // If the Valve is NOT being simulated and it HAS and IS USING limit switch feedback,
   // use the state of the limit switch feedback inputs as the Valve position.
   // If the Valve is being simulated or has no limit switch feedback, use the Sim Timers to provide
   // "fake" feedback signals based on the simulation time to Open and time to Close.
   31: [XIO(Inp_Sim) [XIC(Cfg_UseOpenLS) XIC(Inp_OpenLS) ,XIO(Cfg_UseOpenLS) XIC(Cfg_UseClosedLS) XIO(Inp_ClosedLS) ] ,[XIC(Inp_Sim) ,XIO(Cfg_UseOpenLS) XIO(Cfg_UseClosedLS) ] XIO(Sts_PosInfNaN) GRT(Val_Pos,Cfg_MaxClosedPos) ]OTE(Wrk_OpenFdbk);
   // If the Valve is NOT being simulated and it HAS and IS USING limit switch feedback,
   // use the state of the limit switch feedback inputs as the Valve position.
   // If the Valve is being simulated or has no limit switch feedback, use the Sim Timers to provide
   // "fake" feedback signals based on the simulation time to Open and time to Close.
   32: [XIO(Inp_Sim) [XIC(Cfg_UseClosedLS) XIC(Inp_ClosedLS) ,XIO(Cfg_UseClosedLS) XIC(Cfg_UseOpenLS) XIO(Inp_OpenLS) ] ,[XIC(Inp_Sim) ,XIO(Cfg_UseClosedLS) XIO(Cfg_UseOpenLS) ] XIO(Sts_PosInfNaN) LEQ(Val_Pos,Cfg_MaxClosedPos) ]OTE(Wrk_ClosedFdbk);
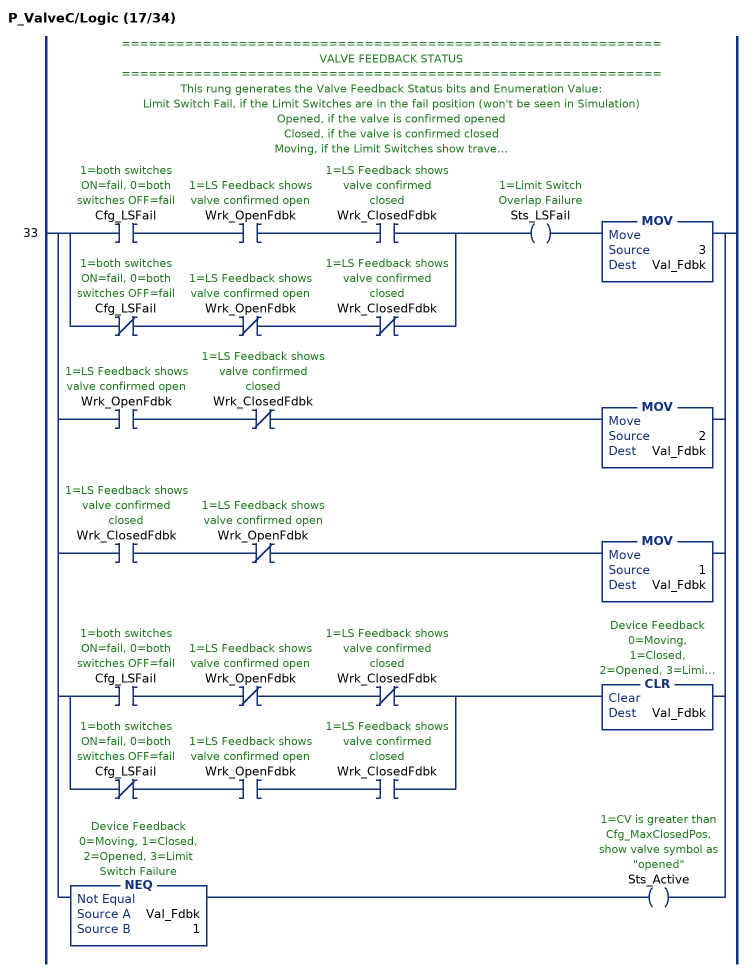
   // ============================================================
   // VALVE FEEDBACK STATUS
   // ============================================================
   // This rung generates the Valve Feedback Status bits and Enumeration Value:
   // Limit Switch Fail, if the Limit Switches are in the fail position (won't be seen in Simulation)
   // Opened, if the valve is confirmed opened
   // Closed, if the valve is confirmed closed
   // Moving, if the Limit Switches show travel
   // If the valve is being reported Open, set the "Active" status (in common with P_PID and
   // P_AOut) to show the analog output graphic symbol on the HMI as "active" (e.g., valve open).
   33: [[XIC(Cfg_LSFail) XIC(Wrk_OpenFdbk) XIC(Wrk_ClosedFdbk) ,XIO(Cfg_LSFail) XIO(Wrk_OpenFdbk) XIO(Wrk_ClosedFdbk) ] OTE(Sts_LSFail) MOV(3,Val_Fdbk) ,XIC(Wrk_OpenFdbk) XIO(Wrk_ClosedFdbk) MOV(2,Val_Fdbk) ,XIC(Wrk_ClosedFdbk) XIO(Wrk_OpenFdbk) MOV(1,Val_Fdbk) ,[XIC(Cfg_LSFail) XIO(Wrk_OpenFdbk) XIO(Wrk_ClosedFdbk) ,XIO(Cfg_LSFail) XIC(Wrk_OpenFdbk) XIC(Wrk_ClosedFdbk) ] CLR(Val_Fdbk) ,NEQ(Val_Fdbk,1) OTE(Sts_Active) ];
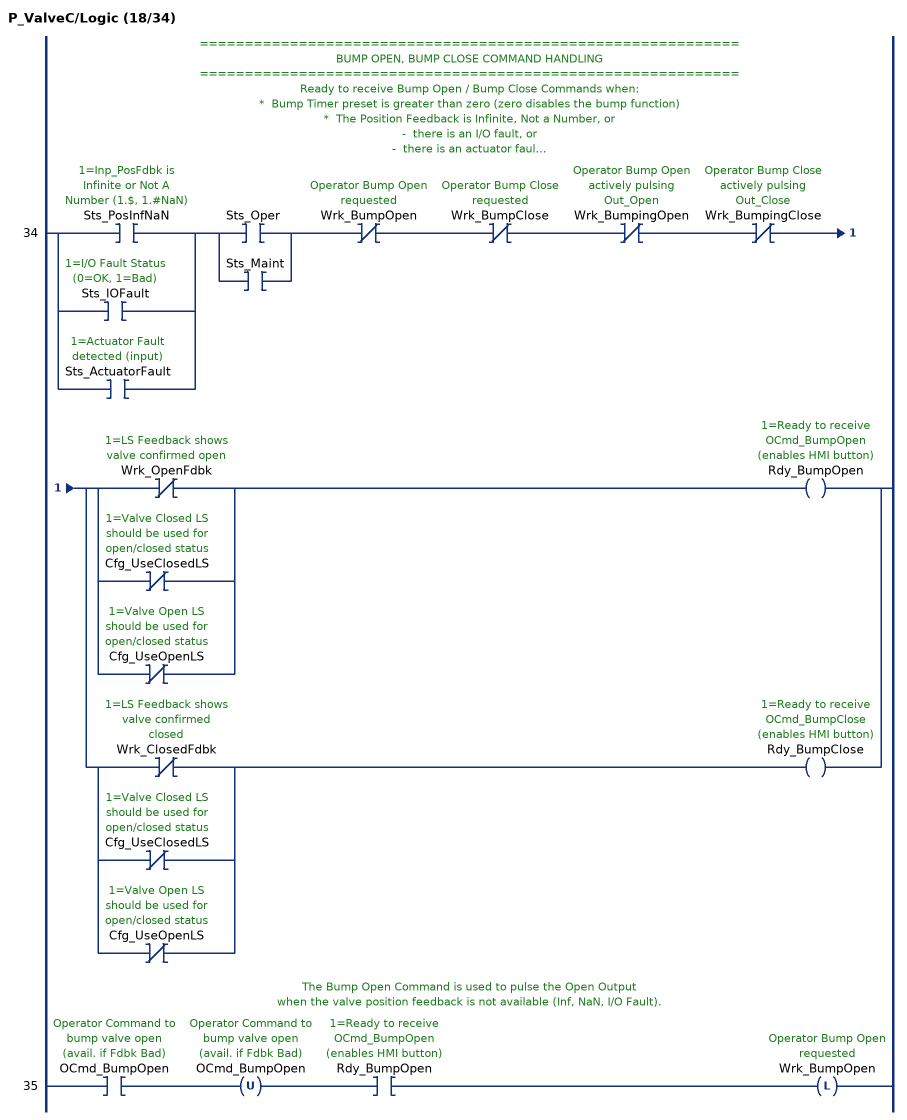
   // ============================================================
   // BUMP OPEN, BUMP CLOSE COMMAND HANDLING
   // ============================================================
   // Ready to receive Bump Open / Bump Close Commands when:
   // *  Bump Timer preset is greater than zero (zero disables the bump function)
   // *  The Position Feedback is Infinite, Not a Number, or
   // -  there is an I/O fault, or
   // -  there is an actuator fault
   // * The valve is in Operator or Maintenance Mode
   // * A previous Bump operation is not active.
   // *  The valve is not at the end of travel (or limit switch is not being used)
   // for the target direction of travel.
   34: [XIC(Sts_PosInfNaN) ,XIC(Sts_IOFault) ,XIC(Sts_ActuatorFault) ][XIC(Sts_Oper) ,XIC(Sts_Maint) ]XIO(Wrk_BumpOpen)XIO(Wrk_BumpClose)XIO(Wrk_BumpingOpen)XIO(Wrk_BumpingClose)[[XIO(Wrk_OpenFdbk) ,XIO(Cfg_UseClosedLS) ,XIO(Cfg_UseOpenLS) ] OTE(Rdy_BumpOpen) ,[XIO(Wrk_ClosedFdbk) ,XIO(Cfg_UseClosedLS) ,XIO(Cfg_UseOpenLS) ] OTE(Rdy_BumpClose) ];
   // The Bump Open Command is used to pulse the Open Output
   // when the valve position feedback is not available (Inf, NaN, I/O Fault).
   35: XIC(OCmd_BumpOpen)OTU(OCmd_BumpOpen)XIC(Rdy_BumpOpen)OTL(Wrk_BumpOpen);
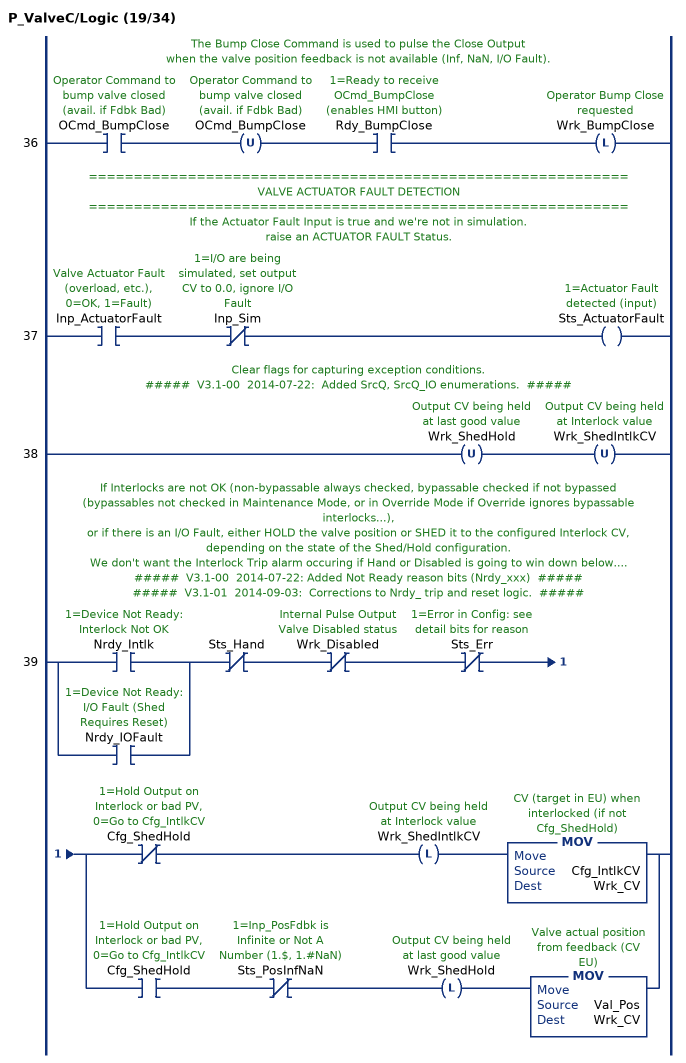
   // The Bump Close Command is used to pulse the Close Output
   // when the valve position feedback is not available (Inf, NaN, I/O Fault).
   36: XIC(OCmd_BumpClose)OTU(OCmd_BumpClose)XIC(Rdy_BumpClose)OTL(Wrk_BumpClose);
   // ============================================================
   // VALVE ACTUATOR FAULT DETECTION
   // ============================================================
   // If the Actuator Fault Input is true and we're not in simulation.
   // raise an ACTUATOR FAULT Status.
   37: XIC(Inp_ActuatorFault)XIO(Inp_Sim)OTE(Sts_ActuatorFault);
   // Clear flags for capturing exception conditions.
   // #####  V3.1-00  2014-07-22:  Added SrcQ, SrcQ_IO enumerations.  #####
   38: OTU(Wrk_ShedHold)OTU(Wrk_ShedIntlkCV);
   // If Interlocks are not OK (non-bypassable always checked, bypassable checked if not bypassed
   // (bypassables not checked in Maintenance Mode, or in Override Mode if Override ignores bypassable interlocks...),
   // or if there is an I/O Fault, either HOLD the valve position or SHED it to the configured Interlock CV,
   // depending on the state of the Shed/Hold configuration.
   // We don't want the Interlock Trip alarm occuring if Hand or Disabled is going to win down below....
   // #####  V3.1-00  2014-07-22: Added Not Ready reason bits (Nrdy_xxx)  #####
   // #####  V3.1-01  2014-09-03:  Corrections to Nrdy_ trip and reset logic.  #####
   39: [XIC(Nrdy_Intlk) ,XIC(Nrdy_IOFault) ]XIO(Sts_Hand)XIO(Wrk_Disabled)XIO(Sts_Err)[XIO(Cfg_ShedHold) OTL(Wrk_ShedIntlkCV) MOV(Cfg_IntlkCV,Wrk_CV) ,XIC(Cfg_ShedHold) XIO(Sts_PosInfNaN) OTL(Wrk_ShedHold) MOV(Val_Pos,Wrk_CV) ];
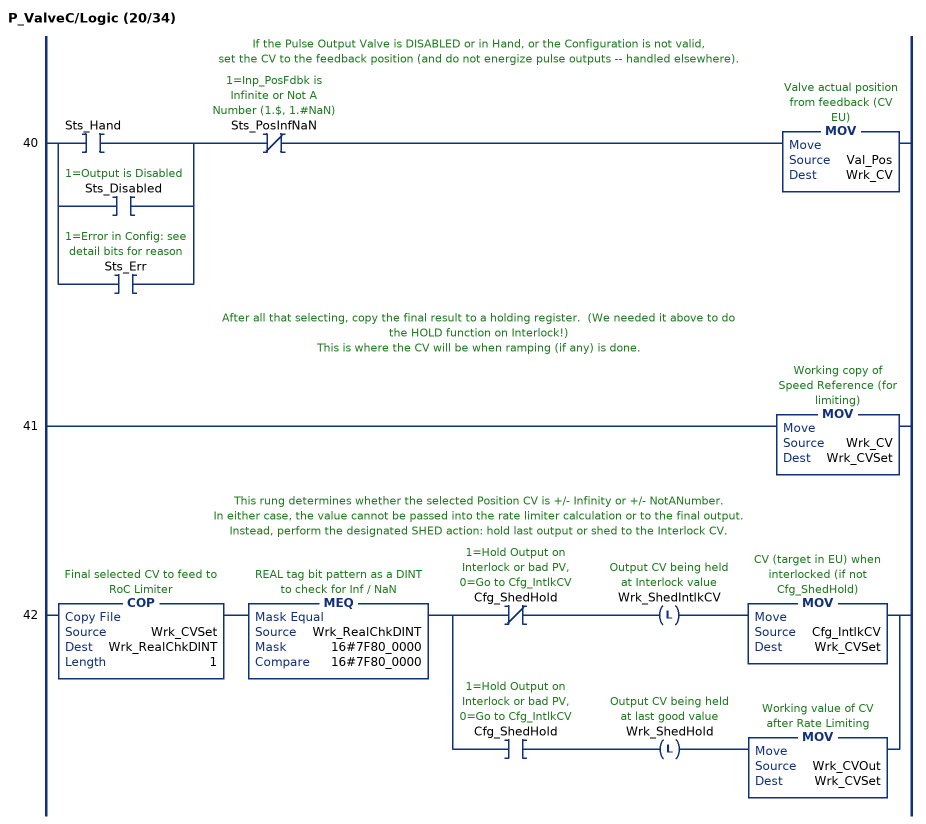
   // If the Pulse Output Valve is DISABLED or in Hand, or the Configuration is not valid,
   // set the CV to the feedback position (and do not energize pulse outputs -- handled elsewhere).
   40: [XIC(Sts_Hand) ,XIC(Sts_Disabled) ,XIC(Sts_Err) ]XIO(Sts_PosInfNaN)MOV(Val_Pos,Wrk_CV);
   // After all that selecting, copy the final result to a holding register.  (We needed it above to do
   // the HOLD function on Interlock!)
   // This is where the CV will be when ramping (if any) is done.
   41: MOV(Wrk_CV,Wrk_CVSet);
   // This rung determines whether the selected Position CV is +/- Infinity or +/- NotANumber.
   // In either case, the value cannot be passed into the rate limiter calculation or to the final output.
   // Instead, perform the designated SHED action: hold last output or shed to the Interlock CV.
   42: COP(Wrk_CVSet,Wrk_RealChkDINT,1)MEQ(Wrk_RealChkDINT,16#7F80_0000,16#7F80_0000)[XIO(Cfg_ShedHold) OTL(Wrk_ShedIntlkCV) MOV(Cfg_IntlkCV,Wrk_CVSet) ,XIC(Cfg_ShedHold) OTL(Wrk_ShedHold) MOV(Wrk_CVOut,Wrk_CVSet) ];
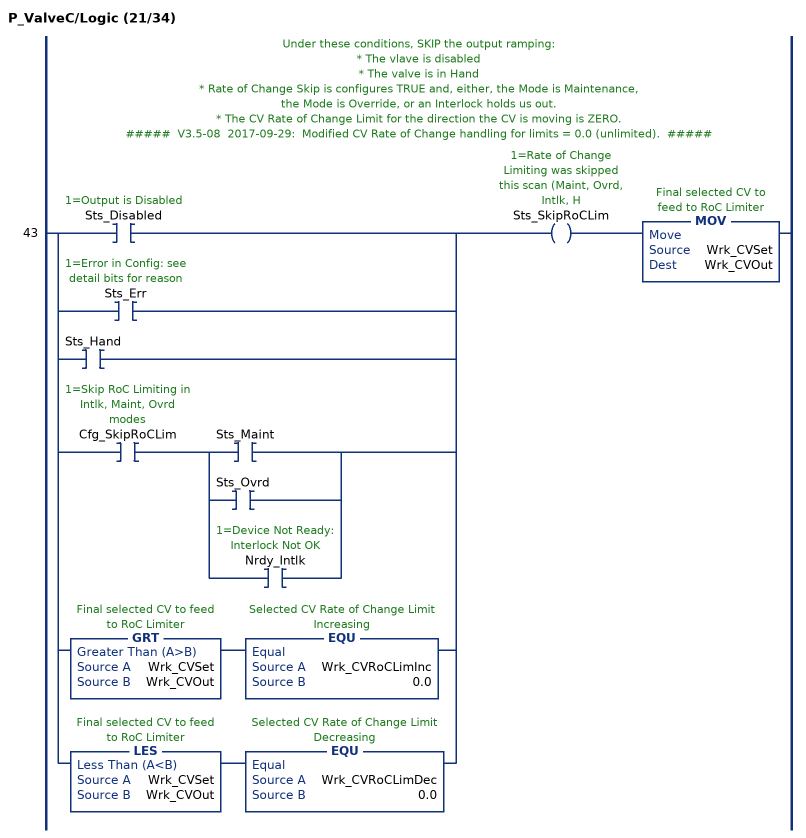
   // Under these conditions, SKIP the output ramping:
   // * The vlave is disabled
   // * The valve is in Hand
   // * Rate of Change Skip is configures TRUE and, either, the Mode is Maintenance,
   // the Mode is Override, or an Interlock holds us out.
   // * The CV Rate of Change Limit for the direction the CV is moving is ZERO.
   // #####  V3.5-08  2017-09-29:  Modified CV Rate of Change handling for limits = 0.0 (unlimited).  #####
   43: [XIC(Sts_Disabled) ,XIC(Sts_Err) ,XIC(Sts_Hand) ,XIC(Cfg_SkipRoCLim) [XIC(Sts_Maint) ,XIC(Sts_Ovrd) ,XIC(Nrdy_Intlk) ] ,GRT(Wrk_CVSet,Wrk_CVOut) EQU(Wrk_CVRoCLimInc,0.0) ,LES(Wrk_CVSet,Wrk_CVOut) EQU(Wrk_CVRoCLimDec,0.0) ]OTE(Sts_SkipRoCLim)MOV(Wrk_CVSet,Wrk_CVOut);
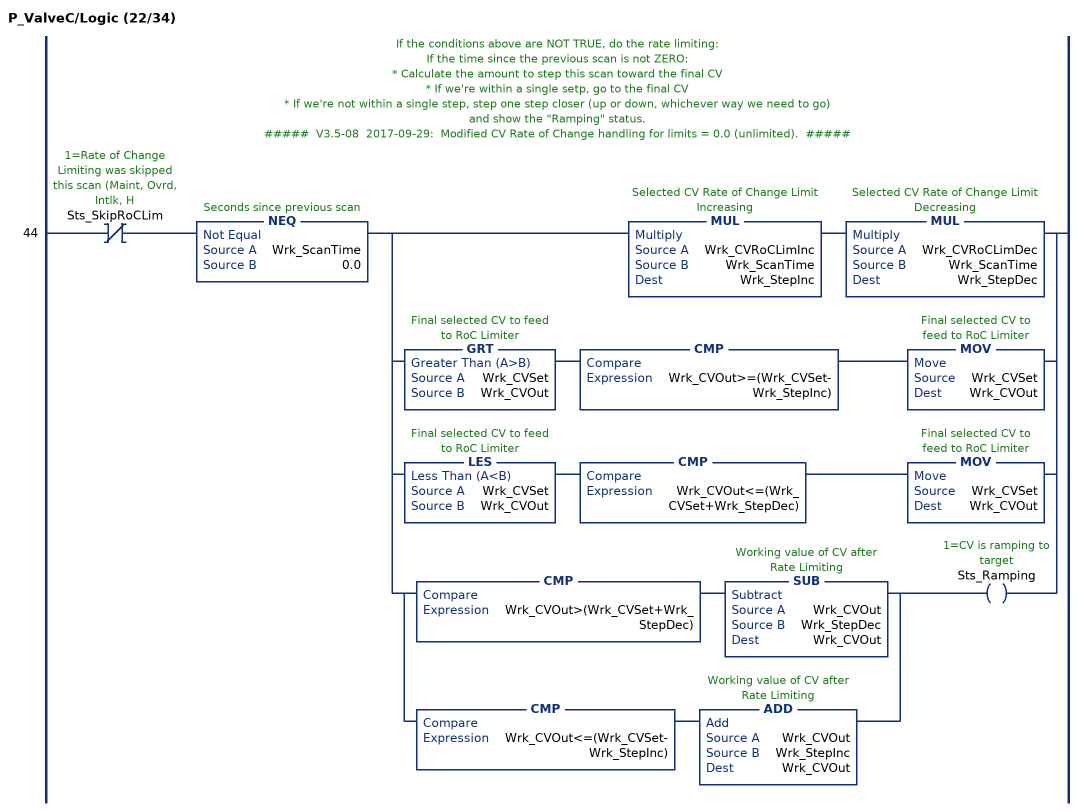
   // If the conditions above are NOT TRUE, do the rate limiting:
   // If the time since the previous scan is not ZERO:
   // * Calculate the amount to step this scan toward the final CV
   // * If we're within a single setp, go to the final CV
   // * If we're not within a single step, step one step closer (up or down, whichever way we need to go)
   // and show the "Ramping" status.
   // #####  V3.5-08  2017-09-29:  Modified CV Rate of Change handling for limits = 0.0 (unlimited).  #####
   44: XIO(Sts_SkipRoCLim)NEQ(Wrk_ScanTime,0.0)[MUL(Wrk_CVRoCLimInc,Wrk_ScanTime,Wrk_StepInc) MUL(Wrk_CVRoCLimDec,Wrk_ScanTime,Wrk_StepDec) ,GRT(Wrk_CVSet,Wrk_CVOut) CMP(Wrk_CVOut>=(Wrk_CVSet-Wrk_StepInc)) MOV(Wrk_CVSet,Wrk_CVOut) ,LES(Wrk_CVSet,Wrk_CVOut) CMP(Wrk_CVOut<=(Wrk_CVSet+Wrk_StepDec)) MOV(Wrk_CVSet,Wrk_CVOut) ,[CMP(Wrk_CVOut>(Wrk_CVSet+Wrk_StepDec)) SUB(Wrk_CVOut,Wrk_StepDec,Wrk_CVOut) ,CMP(Wrk_CVOut<=(Wrk_CVSet-Wrk_StepInc)) ADD(Wrk_CVOut,Wrk_StepInc,Wrk_CVOut) ] OTE(Sts_Ramping) ];
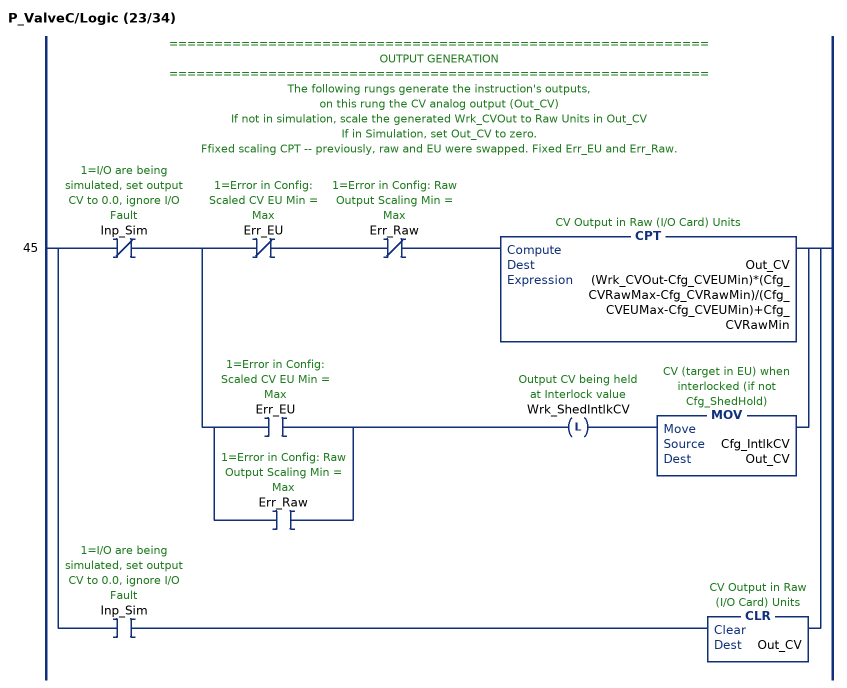
   // ============================================================
   // OUTPUT GENERATION
   // ============================================================
   // The following rungs generate the instruction's outputs,
   // on this rung the CV analog output (Out_CV)
   // If not in simulation, scale the generated Wrk_CVOut to Raw Units in Out_CV
   // If in Simulation, set Out_CV to zero.
   // Ffixed scaling CPT -- previously, raw and EU were swapped. Fixed Err_EU and Err_Raw.
   45: [XIO(Inp_Sim) [XIO(Err_EU) XIO(Err_Raw) CPT(Out_CV,(Wrk_CVOut-Cfg_CVEUMin)*(Cfg_CVRawMax-Cfg_CVRawMin)/(Cfg_CVEUMax-Cfg_CVEUMin)+Cfg_CVRawMin) ,[XIC(Err_EU) ,XIC(Err_Raw) ] OTL(Wrk_ShedIntlkCV) MOV(Cfg_IntlkCV,Out_CV) ] ,XIC(Inp_Sim) CLR(Out_CV) ];
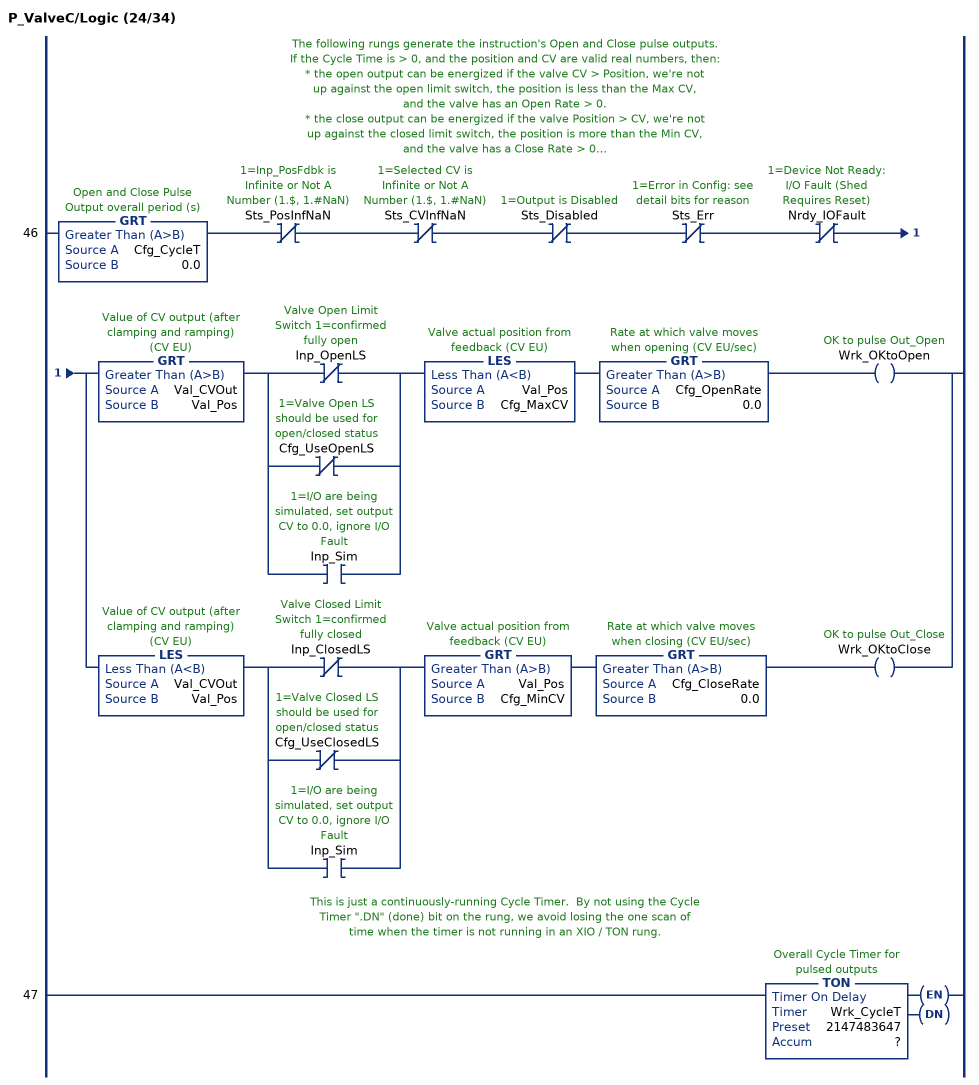
   // The following rungs generate the instruction's Open and Close pulse outputs.
   // If the Cycle Time is > 0, and the position and CV are valid real numbers, then:
   // * the open output can be energized if the valve CV > Position, we're not
   // up against the open limit switch, the position is less than the Max CV,
   // and the valve has an Open Rate > 0.
   // * the close output can be energized if the valve Position > CV, we're not
   // up against the closed limit switch, the position is more than the Min CV,
   // and the valve has a Close Rate > 0.
   // #####  V3.1-03  2015-01-21:  Modified to prevent output pulsing on additional fault conditions.  #####
   46: GRT(Cfg_CycleT,0.0)XIO(Sts_PosInfNaN)XIO(Sts_CVInfNaN)XIO(Sts_Disabled)XIO(Sts_Err)XIO(Nrdy_IOFault)[GRT(Val_CVOut,Val_Pos) [XIO(Inp_OpenLS) ,XIO(Cfg_UseOpenLS) ,XIC(Inp_Sim) ] LES(Val_Pos,Cfg_MaxCV) GRT(Cfg_OpenRate,0.0) OTE(Wrk_OKtoOpen) ,LES(Val_CVOut,Val_Pos) [XIO(Inp_ClosedLS) ,XIO(Cfg_UseClosedLS) ,XIC(Inp_Sim) ] GRT(Val_Pos,Cfg_MinCV) GRT(Cfg_CloseRate,0.0) OTE(Wrk_OKtoClose) ];
   // This is just a continuously-running Cycle Timer.  By not using the Cycle
   // Timer ".DN" (done) bit on the rung, we avoid losing the one scan of
   // time when the timer is not running in an XIO / TON rung.
   47: TON(Wrk_CycleT,?,?);
